LIN {X 0,Y 261.016,Z 653.466,A -85,B 0,C 180,E1 -18954.006,E2 -18954.006} C_VEL
LIN {X 0,Y 257.341,Z 662.24,A -85,B 0,C 180,E1 -18956.893,E2 -18956.893} C_VEL
LIN {X 0,Y 253.986,Z 670.002,A -85,B 0,C 180,E1 -18960.127,E2 -18960.127} C_VEL
LIN {X 0,Y 251.244,Z 676.279,A -85,B 0,C 180,E1 -18963.527,E2 -18963.527} C_VEL
LIN {X 0,Y 249.374,Z 680.762,A -85,B 0,C 180,E1 -18966.762,E2 -18966.762} C_VEL
LIN {X 0,Y 248.037,Z 684.043,A -85,B 0,C 180,E1 -18970.122,E2 -18970.122} C_VEL
LIN {X 0,Y 247.2,Z 686.071,A -85,B 0,C 180,E1 -18973.483,E2 -18973.483} C_VEL
LIN {X 0,Y 246.839,Z 686.909,A -85,B 0,C 180,E1 -18976.834,E2 -18976.834} C_VEL
LIN {X 0,Y 246.696,Z 686.594,A -85,B 0,C 180,E1 -18980.158,E2 -18980.158} C_VEL
LIN {X 0,Y 246.891,Z 685.135,A -85,B 0,C 180,E1 -18983.462,E2 -18983.462} C_VEL
LIN {X 0,Y 247.231,Z 682.514,A -85,B 0,C 180,E1 -18986.741,E2 -18986.741} C_VEL
LIN {X 0,Y 247.801,Z 678.647,A -85,B 0,C 180,E1 -18990,E2 -18990} C_VEL
LIN {X 0,Y 248.772,Z 673.495,A -85,B 0,C 180,E1 -18993.239,E2 -18993.239} C_VEL
LIN {X 0,Y 250.266,Z 666.931,A -85,B 0,C 180,E1 -18996.45,E2 -18996.45} C_VEL
LIN {X 0,Y 252.206,Z 659.844,A -85,B 0,C 180,E1 -18999.22,E2 -18999.22} C_VEL
LIN {X 0,Y 254.44,Z 651.357,A -85,B 0,C 180,E1 -19001.956,E2 -19001.956} C_VEL
LIN {X 0,Y 257.158,Z 641.157,A -85,B 0,C 180,E1 -19004.643,E2 -19004.643} C_VEL
LIN {X 0,Y 259.96,Z 630.71,A -85,B 0,C 180,E1 -19006.896,E2 -19006.896} C_VEL
LIN {X 0,Y 262.686,Z 619.377,A -85,B 0,C 180,E1 -19008.929,E2 -19008.929} C_VEL
LIN {X 0,Y 265.451,Z 607.068,A -85,B 0,C 180,E1 -19010.739,E2 -19010.739} C_VEL
LIN {X 0,Y 268.125,Z 593.612,A -85,B 0,C 180,E1 -19012.338,E2 -19012.338} C_VEL
LIN {X 0,Y 270.433,Z 579.688,A -85,B 0,C 180,E1 -19013.653,E2 -19013.653} C_VEL
LIN {X 0,Y 272.361,Z 565.38,A -85,B 0,C 180,E1 -19014.69,E2 -19014.69} C_VEL
LIN {X 0,Y 273.951,Z 549.877,A -85,B 0,C 180,E1 -19015.5,E2 -19015.5} C_VEL
LIN {X 0,Y 274.904,Z 534.682,A -85,B 0,C 180,E1 -19016.017,E2 -19016.017} C_VEL
LIN {X 0,Y 279.025,Z 439.219,A -85,B 0,C 180,E1 -19018.376,E2 -19018.376} C_VEL
LIN {X 0,Y 272.382,Z 423.601,A -85,B 0,C 180,E1 -19019.845,E2 -19019.845} C_VEL
LIN {X 0,Y 268.047,Z 414.836,A -85,B 0,C 180,E1 -19020.812,E2 -19020.812} C_VEL
LIN {X 0,Y 259.634,Z 400.449,A -85,B 0,C 180,E1 -19022.72,E2 -19022.72} C_VEL
LIN {X 0,Y 253.489,Z 390.868,A -85,B 0,C 180,E1 -19024.195,E2 -19024.195} C_VEL
LIN {X 0,Y 251.182,Z 387.293,A -85,B 0,C 180,E1 -19024.776,E2 -19024.776} C_VEL
LIN {X 0,Y 249.581,Z 385.053,A -85,B 0,C 180,E1 -19025.178,E2 -19025.178} C_VEL
LIN {X 0,Y 249.044,Z 383.079,A -85,B 0,C 180,E1 -19025.377,E2 -19025.377} C_VEL
LIN {X 0,Y 249.025,Z 383.091,A -85,B 0,C 180,E1 -19028.381,E2 -19028.381} C_VEL
LIN {X 0,Y 248.997,Z 383.093,A -85,B 0,C 180,E1 -19032.788,E2 -19032.788} C_VEL
LIN {X 0,Y 248.982,Z 383.08,A -85,B 0,C 180,E1 -19037.354,E2 -19037.354} C_VEL
LIN {X 0,Y 249.024,Z 383.085,A -85,B 0,C 180,E1 -19042.207,E2 -19042.207} C_VEL
LIN {X 0,Y 249.045,Z 383.078,A -85,B 0,C 180,E1 -19045.639,E2 -19045.639} C_VEL
LIN {X 0,Y 249.004,Z 383.09,A -85,B 0,C 180,E1 -19049.466,E2 -19049.466} C_VEL
LIN {X 0,Y 249.014,Z 383.029,A -85,B 0,C 180,E1 -19053.154,E2 -19053.154} C_VEL
LIN {X 0,Y 249.01,Z 383.065,A -85,B 0,C 180,E1 -19056.725,E2 -19056.725} C_VEL
LIN {X 0,Y 249.088,Z 383.08,A -85,B 0,C 180,E1 -19060.209,E2 -19060.209} C_VEL
LIN {X 0,Y 249.198,Z 383.054,A -85,B 0,C 180,E1 -19063.618,E2 -19063.618} C_VEL
LIN {X 0,Y 249.19,Z 383.049,A -85,B 0,C 180,E1 -19067.817,E2 -19067.817} C_VEL
LIN {X 0,Y 248.56,Z 383.129,A -85,B 0,C 180,E1 -19069.168,E2 -19069.168} C_VEL
LIN {X 0,Y 245.742,Z 383.496,A -85,B 0,C 180,E1 -19071.372,E2 -19071.372} C_VEL
LIN {X 0,Y 243.333,Z 383.789,A -85,B 0,C 180,E1 -19073.167,E2 -19073.167} C_VEL
LIN {X 0,Y 242.305,Z 383.906,A -85,B 0,C 180,E1 -19074.558,E2 -19074.558} C_VEL
LIN {X 0,Y 242.225,Z 383.914,A -85,B 0,C 180,E1 -19075.03,E2 -19075.03} C_VEL
LIN {X 0,Y 242.622,Z 383.886,A -85,B 0,C 180,E1 -19078.339,E2 -19078.339} C_VEL
LIN {X 0,Y 242.624,Z 383.866,A -85,B 0,C 180,E1 -19081.659,E2 -19081.659} C_VEL
LIN {X 0,Y 242.4,Z 383.906,A -85,B 0,C 180,E1 -19086.659,E2 -19086.659} C_VEL
LIN {X 0,Y 242.266,Z 383.931,A -85,B 0,C 180,E1 -19090.023,E2 -19090.023} C_VEL
LIN {X 0,Y 242.114,Z 383.946,A -85,B 0,C 180,E1 -19095.144,E2 -19095.144} C_VEL
LIN {X 0,Y 242.055,Z 383.945,A -85,B 0,C 180,E1 -19098.625,E2 -19098.625} C_VEL
LIN {X 0,Y 242.006,Z 383.951,A -85,B 0,C 180,E1 -19102.18,E2 -19102.18} C_VEL
LIN {X 0,Y 242.033,Z 383.952,A -85,B 0,C 180,E1 -19105.82,E2 -19105.82} C_VEL
LIN {X 0,Y 241.969,Z 383.963,A -85,B 0,C 180,E1 -19109.588,E2 -19109.588} C_VEL
LIN {X 0,Y 241.979,Z 383.964,A -85,B 0,C 180,E1 -19113.492,E2 -19113.492} C_VEL
LIN {X 0,Y 241.964,Z 383.967,A -85,B 0,C 180,E1 -19117.586,E2 -19117.586} C_VEL
LIN {X 0,Y 241.953,Z 384.049,A -85,B 0,C 180,E1 -19121.289,E2 -19121.289} C_VEL
LIN {X 0,Y 243.383,Z 388.779,A -85,B 0,C 180,E1 -19123.277,E2 -19123.277} C_VEL
LIN {X 0,Y 251.725,Z 403.288,A -85,B 0,C 180,E1 -19125.515,E2 -19125.515} C_VEL
LIN {X 0,Y 259.948,Z 419.151,A -85,B 0,C 180,E1 -19127.579,E2 -19127.579} C_VEL
LIN {X 0,Y 266.809,Z 434.583,A -85,B 0,C 180,E1 -19129.238,E2 -19129.238} C_VEL
LIN {X 0,Y 271.986,Z 447.57,A -85,B 0,C 180,E1 -19130.456,E2 -19130.456} C_VEL
LIN {X 0,Y 272.722,Z 452.165,A -85,B 0,C 180,E1 -19130.712,E2 -19130.712} C_VEL
LIN {X 0,Y 268.172,Z 555.027,A -85,B 0,C 180,E1 -19133.342,E2 -19133.342} C_VEL
LIN {X 0,Y 266.741,Z 570.811,A -85,B 0,C 180,E1 -19133.993,E2 -19133.993} C_VEL
LIN {X 0,Y 264.605,Z 586.544,A -85,B 0,C 180,E1 -19134.944,E2 -19134.944} C_VEL
LIN {X 0,Y 262.082,Z 601.542,A -85,B 0,C 180,E1 -19136.196,E2 -19136.196} C_VEL
LIN {X 0,Y 259.354,Z 615.018,A -85,B 0,C 180,E1 -19137.643,E2 -19137.643} C_VEL
LIN {X 0,Y 256.193,Z 628.75,A -85,B 0,C 180,E1 -19139.502,E2 -19139.502} C_VEL
LIN {X 0,Y 253.314,Z 640.146,A -85,B 0,C 180,E1 -19141.407,E2 -19141.407} C_VEL
LIN {X 0,Y 250.333,Z 651.665,A -85,B 0,C 180,E1 -19143.758,E2 -19143.758} C_VEL
LIN {X 0,Y 247.409,Z 662.845,A -85,B 0,C 180,E1 -19146.566,E2 -19146.566} C_VEL
LIN {X 0,Y 244.839,Z 672.073,A -85,B 0,C 180,E1 -19149.413,E2 -19149.413} C_VEL
LIN {X 0,Y 242.894,Z 679.934,A -85,B 0,C 180,E1 -19152.4,E2 -19152.4} C_VEL
LIN {X 0,Y 241.36,Z 686.864,A -85,B 0,C 180,E1 -19155.67,E2 -19155.67} C_VEL
LIN {X 0,Y 240.349,Z 692.458,A -85,B 0,C 180,E1 -19159.043,E2 -19159.043} C_VEL
LIN {X 0,Y 240.014,Z 695.768,A -85,B 0,C 180,E1 -19161.581,E2 -19161.581} C_VEL
LIN {X 0,Y 239.835,Z 699.127,A -85,B 0,C 180,E1 -19165.077,E2 -19165.077} C_VEL
LIN {X 0,Y 239.871,Z 701.027,A -85,B 0,C 180,E1 -19168.321,E2 -19168.321} C_VEL
LIN {X 0,Y 239.924,Z 701.581,A -85,B 0,C 180,E1 -19170,E2 -19170} C_VEL
LIN {X 0,Y 239.761,Z 701.819,A -85,B 0,C 180,E1 -19173.361,E2 -19173.361} C_VEL
LIN {X 0,Y 239.788,Z 700.928,A -85,B 0,C 180,E1 -19176.733,E2 -19176.733} C_VEL
LIN {X 0,Y 240.257,Z 698.904,A -85,B 0,C 180,E1 -19180.108,E2 -19180.108} C_VEL
LIN {X 0,Y 241.291,Z 695.662,A -85,B 0,C 180,E1 -19183.474,E2 -19183.474} C_VEL
LIN {X 0,Y 242.893,Z 691.191,A -85,B 0,C 180,E1 -19186.819,E2 -19186.819} C_VEL
LIN {X 0,Y 245.272,Z 685.389,A -85,B 0,C 180,E1 -19190.111,E2 -19190.111} C_VEL
LIN {X 0,Y 248.318,Z 678.108,A -85,B 0,C 180,E1 -19193.343,E2 -19193.343} C_VEL
LIN {X 0,Y 251.8,Z 670.353,A -85,B 0,C 180,E1 -19196.078,E2 -19196.078} C_VEL
LIN {X 0,Y 254.976,Z 662.549,A -85,B 0,C 180,E1 -19198.39,E2 -19198.39} C_VEL
LIN {X 0,Y 259.415,Z 651.682,A -85,B 0,C 180,E1 -19200.98,E2 -19200.98} C_VEL
LIN {X 0,Y 263.606,Z 640.549,A -85,B 0,C 180,E1 -19203.131,E2 -19203.131} C_VEL
LIN {X 0,Y 267.847,Z 628.357,A -85,B 0,C 180,E1 -19205.028,E2 -19205.028} C_VEL
LIN {X 0,Y 270.967,Z 618.154,A -85,B 0,C 180,E1 -19206.335,E2 -19206.335} C_VEL
LIN {X 0,Y 274.472,Z 605.361,A -85,B 0,C 180,E1 -19207.686,E2 -19207.686} C_VEL
LIN {X 0,Y 277.752,Z 590.92,A -85,B 0,C 180,E1 -19208.891,E2 -19208.891} C_VEL
LIN {X 0,Y 280.638,Z 575.825,A -85,B 0,C 180,E1 -19209.804,E2 -19209.804} C_VEL
LIN {X 0,Y 282.692,Z 560.992,A -85,B 0,C 180,E1 -19210.445,E2 -19210.445} C_VEL
LIN {X 0,Y 283.971,Z 544.545,A -85,B 0,C 180,E1 -19210.925,E2 -19210.925} C_VEL
LIN {X 0,Y 288.516,Z 461.824,A -85,B 0,C 180,E1 -19212.922,E2 -19212.922} C_VEL
LIN {X 0,Y 282.932,Z 449.608,A -85,B 0,C 180,E1 -19214.599,E2 -19214.599} C_VEL
LIN {X 0,Y 277.69,Z 439.213,A -85,B 0,C 180,E1 -19216.25,E2 -19216.25} C_VEL
LIN {X 0,Y 270.529,Z 426.425,A -85,B 0,C 180,E1 -19218.661,E2 -19218.661} C_VEL
LIN {X 0,Y 263.822,Z 415.704,A -85,B 0,C 180,E1 -19221.121,E2 -19221.121} C_VEL
LIN {X 0,Y 259.64,Z 409.46,A -85,B 0,C 180,E1 -19222.783,E2 -19222.783} C_VEL
LIN {X 0,Y 256.451,Z 404.711,A -85,B 0,C 180,E1 -19224.143,E2 -19224.143} C_VEL
LIN {X 0,Y 252.023,Z 398.57,A -85,B 0,C 180,E1 -19226.166,E2 -19226.166} C_VEL
LIN {X 0,Y 248.403,Z 393.715,A -85,B 0,C 180,E1 -19227.967,E2 -19227.967} C_VEL
LIN {X 0,Y 246.962,Z 391.993,A -85,B 0,C 180,E1 -19228.717,E2 -19228.717} C_VEL
LIN {X 0,Y 244,Z 388.202,A -85,B 0,C 180,E1 -19230.369,E2 -19230.369} C_VEL
LIN {X 0,Y 242.753,Z 386.342,A -85,B 0,C 180,E1 -19231.167,E2 -19231.167} C_VEL
LIN {X 0,Y 241.997,Z 383.957,A -85,B 0,C 180,E1 -19233.248,E2 -19233.248} C_VEL
LIN {X 0,Y 242.027,Z 383.957,A -85,B 0,C 180,E1 -19236.013,E2 -19236.013} C_VEL
LIN {X 0,Y 242.036,Z 383.955,A -85,B 0,C 180,E1 -19239.609,E2 -19239.609} C_VEL
LIN {X 0,Y 242.164,Z 383.937,A -85,B 0,C 180,E1 -19243.279,E2 -19243.279} C_VEL
LIN {X 0,Y 242.151,Z 383.942,A -85,B 0,C 180,E1 -19246.575,E2 -19246.575} C_VEL
LIN {X 0,Y 242.343,Z 383.918,A -85,B 0,C 180,E1 -19250.405,E2 -19250.405} C_VEL
LIN {X 0,Y 242.399,Z 383.915,A -85,B 0,C 180,E1 -19253.341,E2 -19253.341} C_VEL
LIN {X 0,Y 242.631,Z 383.882,A -85,B 0,C 180,E1 -19258.341,E2 -19258.341} C_VEL
LIN {X 0,Y 242.624,Z 383.889,A -85,B 0,C 180,E1 -19261.661,E2 -19261.661} C_VEL
LIN {X 0,Y 242.4,Z 383.906,A -85,B 0,C 180,E1 -19266.661,E2 -19266.661} C_VEL
LIN {X 0,Y 242.27,Z 383.926,A -85,B 0,C 180,E1 -19270.024,E2 -19270.024} C_VEL
LIN {X 0,Y 242.169,Z 383.935,A -85,B 0,C 180,E1 -19275.141,E2 -19275.141} C_VEL
LIN {X 0,Y 242.051,Z 383.922,A -85,B 0,C 180,E1 -19278.791,E2 -19278.791} C_VEL
LIN {X 0,Y 242.765,Z 386.257,A -85,B 0,C 180,E1 -19279.337,E2 -19279.337} C_VEL
LIN {X 0,Y 244.854,Z 388.758,A -85,B 0,C 180,E1 -19280.555,E2 -19280.555} C_VEL
LIN {X 0,Y 246.633,Z 389.798,A -85,B 0,C 180,E1 -19281.462,E2 -19281.462} C_VEL
LIN {X 0,Y 248.217,Z 392.799,A -85,B 0,C 180,E1 -19282.364,E2 -19282.364} C_VEL
LIN {X 0,Y 250.878,Z 395.128,A -85,B 0,C 180,E1 -19283.638,E2 -19283.638} C_VEL
LIN {X 0,Y 253.737,Z 399.159,A -85,B 0,C 180,E1 -19285.009,E2 -19285.009} C_VEL
LIN {X 0,Y 255.513,Z 400.971,A -85,B 0,C 180,E1 -19285.782,E2 -19285.782} C_VEL
LIN {X 0,Y 258.133,Z 404.484,A -85,B 0,C 180,E1 -19286.914,E2 -19286.914} C_VEL
LIN {X 0,Y 259.914,Z 406.69,A -85,B 0,C 180,E1 -19287.64,E2 -19287.64} C_VEL
LIN {X 0,Y 263.34,Z 411.23,A -85,B 0,C 180,E1 -19288.984,E2 -19288.984} C_VEL
LIN {X 0,Y 269.38,Z 419.469,A -85,B 0,C 180,E1 -19291.18,E2 -19291.18} C_VEL
LIN {X 0,Y 276.643,Z 430.325,A -85,B 0,C 180,E1 -19293.598,E2 -19293.598} C_VEL
LIN {X 0,Y 282.542,Z 440.74,A -85,B 0,C 180,E1 -19295.443,E2 -19295.443} C_VEL
LIN {X 0,Y 288.955,Z 453.487,A -85,B 0,C 180,E1 -19297.34,E2 -19297.34} C_VEL
LIN {X 0,Y 283.774,Z 541.587,A -85,B 0,C 180,E1 -19299.44,E2 -19299.44} C_VEL
LIN {X 0,Y 282.258,Z 556.763,A -85,B 0,C 180,E1 -19300.037,E2 -19300.037} C_VEL
LIN {X 0,Y 280.123,Z 570.776,A -85,B 0,C 180,E1 -19300.813,E2 -19300.813} C_VEL
LIN {X 0,Y 277.323,Z 585.198,A -85,B 0,C 180,E1 -19301.89,E2 -19301.89} C_VEL
LIN {X 0,Y 274.227,Z 597.838,A -85,B 0,C 180,E1 -19303.079,E2 -19303.079} C_VEL
LIN {X 0,Y 270.778,Z 610.647,A -85,B 0,C 180,E1 -19304.621,E2 -19304.621} C_VEL
LIN {X 0,Y 267.002,Z 622.242,A -85,B 0,C 180,E1 -19306.295,E2 -19306.295} C_VEL
LIN {X 0,Y 262.9,Z 633.747,A -85,B 0,C 180,E1 -19308.349,E2 -19308.349} C_VEL
LIN {X 0,Y 259.167,Z 643.251,A -85,B 0,C 180,E1 -19310.412,E2 -19310.412} C_VEL
LIN {X 0,Y 255.07,Z 653.132,A -85,B 0,C 180,E1 -19313.04,E2 -19313.04} C_VEL
LIN {X 0,Y 251.163,Z 661.982,A -85,B 0,C 180,E1 -19315.969,E2 -19315.969} C_VEL
LIN {X 0,Y 247.592,Z 669.859,A -85,B 0,C 180,E1 -19319.274,E2 -19319.274} C_VEL
LIN {X 0,Y 244.737,Z 676.055,A -85,B 0,C 180,E1 -19322.648,E2 -19322.648} C_VEL
LIN {X 0,Y 242.606,Z 680.758,A -85,B 0,C 180,E1 -19326.074,E2 -19326.074} C_VEL
LIN {X 0,Y 241.135,Z 684.108,A -85,B 0,C 180,E1 -19329.528,E2 -19329.528} C_VEL
LIN {X 0,Y 240.196,Z 686.207,A -85,B 0,C 180,E1 -19332.987,E2 -19332.987} C_VEL
LIN {X 0,Y 239.783,Z 687.114,A -85,B 0,C 180,E1 -19336.439,E2 -19336.439} C_VEL
LIN {X 0,Y 239.605,Z 686.867,A -85,B 0,C 180,E1 -19339.864,E2 -19339.864} C_VEL
LIN {X 0,Y 239.773,Z 685.477,A -85,B 0,C 180,E1 -19343.267,E2 -19343.267} C_VEL
LIN {X 0,Y 239.973,Z 684.337,A -85,B 0,C 180,E1 -19344.96,E2 -19344.96} C_VEL
LIN {X 0,Y 240.325,Z 681.149,A -85,B 0,C 180,E1 -19348.324,E2 -19348.324} C_VEL
LIN {X 0,Y 241.158,Z 676.72,A -85,B 0,C 180,E1 -19351.67,E2 -19351.67} C_VEL
LIN {X 0,Y 242.427,Z 670.96,A -85,B 0,C 180,E1 -19354.989,E2 -19354.989} C_VEL
LIN {X 0,Y 244.271,Z 663.702,A -85,B 0,C 180,E1 -19358.271,E2 -19358.271} C_VEL
LIN {X 0,Y 246.499,Z 655.924,A -85,B 0,C 180,E1 -19361.096,E2 -19361.096} C_VEL
LIN {X 0,Y 249.079,Z 646.608,A -85,B 0,C 180,E1 -19363.877,E2 -19363.877} C_VEL
LIN {X 0,Y 251.693,Z 637.137,A -85,B 0,C 180,E1 -19366.214,E2 -19366.214} C_VEL
LIN {X 0,Y 254.743,Z 625.879,A -85,B 0,C 180,E1 -19368.498,E2 -19368.498} C_VEL
LIN {X 0,Y 257.723,Z 613.535,A -85,B 0,C 180,E1 -19370.555,E2 -19370.555} C_VEL
LIN {X 0,Y 260.701,Z 599.893,A -85,B 0,C 180,E1 -19372.382,E2 -19372.382} C_VEL
LIN {X 0,Y 263.204,Z 586.496,A -85,B 0,C 180,E1 -19373.82,E2 -19373.82} C_VEL
LIN {X 0,Y 265.467,Z 571.622,A -85,B 0,C 180,E1 -19375.061,E2 -19375.061} C_VEL
LIN {X 0,Y 267.314,Z 556.746,A -85,B 0,C 180,E1 -19375.971,E2 -19375.971} C_VEL
LIN {X 0,Y 268.538,Z 541.777,A -85,B 0,C 180,E1 -19376.613,E2 -19376.613} C_VEL
LIN {X 0,Y 273.103,Z 442.016,A -85,B 0,C 180,E1 -19379.148,E2 -19379.148} C_VEL
LIN {X 0,Y 272.682,Z 440.051,A -85,B 0,C 180,E1 -19379.274,E2 -19379.274} C_VEL
LIN {X 0,Y 265.883,Z 424.291,A -85,B 0,C 180,E1 -19380.848,E2 -19380.848} C_VEL
LIN {X 0,Y 259.43,Z 412.346,A -85,B 0,C 180,E1 -19382.341,E2 -19382.341} C_VEL
LIN {X 0,Y 251.681,Z 399.57,A -85,B 0,C 180,E1 -19384.223,E2 -19384.223} C_VEL
LIN {X 0,Y 246.829,Z 392.184,A -85,B 0,C 180,E1 -19385.467,E2 -19385.467} C_VEL
LIN {X 0,Y 244.256,Z 388.333,A -85,B 0,C 180,E1 -19386.151,E2 -19386.151} C_VEL
LIN {X 0,Y 242.488,Z 385.859,A -85,B 0,C 180,E1 -19386.628,E2 -19386.628} C_VEL
LIN {X 0,Y 241.977,Z 383.956,A -85,B 0,C 180,E1 -19386.854,E2 -19386.854} C_VEL
LIN {X 0,Y 241.917,Z 383.957,A -85,B 0,C 180,E1 -19390.944,E2 -19390.944} C_VEL
LIN {X 0,Y 241.914,Z 383.967,A -85,B 0,C 180,E1 -19394.206,E2 -19394.206} C_VEL
LIN {X 0,Y 241.909,Z 383.97,A -85,B 0,C 180,E1 -19398.07,E2 -19398.07} C_VEL
LIN {X 0,Y 241.968,Z 383.965,A -85,B 0,C 180,E1 -19402.413,E2 -19402.413} C_VEL
LIN {X 0,Y 241.982,Z 383.959,A -85,B 0,C 180,E1 -19406.507,E2 -19406.507} C_VEL
LIN {X 0,Y 241.978,Z 383.947,A -85,B 0,C 180,E1 -19410.613,E2 -19410.613} C_VEL
LIN {X 0,Y 241.998,Z 383.901,A -85,B 0,C 180,E1 -19414.197,E2 -19414.197} C_VEL
LIN {X 0,Y 242.018,Z 383.96,A -85,B 0,C 180,E1 -19418.319,E2 -19418.319} C_VEL
LIN {X 0,Y 242.118,Z 383.933,A -85,B 0,C 180,E1 -19423.315,E2 -19423.315} C_VEL
LIN {X 0,Y 242.142,Z 383.927,A -85,B 0,C 180,E1 -19427.836,E2 -19427.836} C_VEL
LIN {X 0,Y 242.387,Z 383.916,A -85,B 0,C 180,E1 -19431.663,E2 -19431.663} C_VEL
LIN {X 0,Y 242.403,Z 383.903,A -85,B 0,C 180,E1 -19433.34,E2 -19433.34} C_VEL
LIN {X 0,Y 242.225,Z 383.914,A -85,B 0,C 180,E1 -19435.03,E2 -19435.03} C_VEL
LIN {X 0,Y 241.632,Z 383.999,A -85,B 0,C 180,E1 -19436.422,E2 -19436.422} C_VEL
LIN {X 0,Y 239.015,Z 384.335,A -85,B 0,C 180,E1 -19438.701,E2 -19438.701} C_VEL
LIN {X 0,Y 235.856,Z 384.71,A -85,B 0,C 180,E1 -19441.503,E2 -19441.503} C_VEL
LIN {X 0,Y 235.424,Z 384.765,A -85,B 0,C 180,E1 -19442.47,E2 -19442.47} C_VEL
LIN {X 0,Y 235.351,Z 384.782,A -85,B 0,C 180,E1 -19446.859,E2 -19446.859} C_VEL
LIN {X 0,Y 235.212,Z 384.809,A -85,B 0,C 180,E1 -19450.327,E2 -19450.327} C_VEL
LIN {X 0,Y 235.065,Z 384.827,A -85,B 0,C 180,E1 -19455.609,E2 -19455.609} C_VEL
LIN {X 0,Y 234.996,Z 384.828,A -85,B 0,C 180,E1 -19459.206,E2 -19459.206} C_VEL
LIN {X 0,Y 234.948,Z 384.831,A -85,B 0,C 180,E1 -19462.883,E2 -19462.883} C_VEL
LIN {X 0,Y 234.945,Z 384.835,A -85,B 0,C 180,E1 -19466.66,E2 -19466.66} C_VEL
LIN {X 0,Y 234.899,Z 384.846,A -85,B 0,C 180,E1 -19470.572,E2 -19470.572} C_VEL
LIN {X 0,Y 234.921,Z 384.848,A -85,B 0,C 180,E1 -19474.639,E2 -19474.639} C_VEL
LIN {X 0,Y 234.9,Z 384.831,A -85,B 0,C 180,E1 -19479.476,E2 -19479.476} C_VEL
LIN {X 0,Y 234.902,Z 384.921,A -85,B 0,C 180,E1 -19480.033,E2 -19480.033} C_VEL
LIN {X 0,Y 236.055,Z 388.638,A -85,B 0,C 180,E1 -19481.632,E2 -19481.632} C_VEL
LIN {X 0,Y 242.869,Z 400.164,A -85,B 0,C 180,E1 -19483.614,E2 -19483.614} C_VEL
LIN {X 0,Y 248.037,Z 409.511,A -85,B 0,C 180,E1 -19485.029,E2 -19485.029} C_VEL
LIN {X 0,Y 255.154,Z 423.383,A -85,B 0,C 180,E1 -19486.88,E2 -19486.88} C_VEL
LIN {X 0,Y 261.861,Z 438.74,A -85,B 0,C 180,E1 -19488.573,E2 -19488.573} C_VEL
LIN {X 0,Y 266.476,Z 450.566,A -85,B 0,C 180,E1 -19489.711,E2 -19489.711} C_VEL
LIN {X 0,Y 266.886,Z 454.888,A -85,B 0,C 180,E1 -19489.916,E2 -19489.916} C_VEL
LIN {X 0,Y 262.175,Z 555.901,A -85,B 0,C 180,E1 -19492.542,E2 -19492.542} C_VEL
LIN {X 0,Y 260.688,Z 571.263,A -85,B 0,C 180,E1 -19493.201,E2 -19493.201} C_VEL
LIN {X 0,Y 258.577,Z 586.173,A -85,B 0,C 180,E1 -19494.122,E2 -19494.122} C_VEL
LIN {X 0,Y 256.163,Z 600.234,A -85,B 0,C 180,E1 -19495.304,E2 -19495.304} C_VEL
LIN {X 0,Y 253.337,Z 613.909,A -85,B 0,C 180,E1 -19496.777,E2 -19496.777} C_VEL
LIN {X 0,Y 250.012,Z 627.824,A -85,B 0,C 180,E1 -19498.664,E2 -19498.664} C_VEL
LIN {X 0,Y 247.101,Z 639.327,A -85,B 0,C 180,E1 -19500.618,E2 -19500.618} C_VEL
LIN {X 0,Y 243.909,Z 650.749,A -85,B 0,C 180,E1 -19502.964,E2 -19502.964} C_VEL
LIN {X 0,Y 241.231,Z 660.698,A -85,B 0,C 180,E1 -19505.471,E2 -19505.471} C_VEL
LIN {X 0,Y 238.461,Z 670.255,A -85,B 0,C 180,E1 -19508.383,E2 -19508.383} C_VEL
LIN {X 0,Y 236.36,Z 678.203,A -85,B 0,C 180,E1 -19511.358,E2 -19511.358} C_VEL
LIN {X 0,Y 234.752,Z 684.78,A -85,B 0,C 180,E1 -19514.369,E2 -19514.369} C_VEL
LIN {X 0,Y 233.503,Z 690.802,A -85,B 0,C 180,E1 -19517.837,E2 -19517.837} C_VEL
LIN {X 0,Y 232.941,Z 695.426,A -85,B 0,C 180,E1 -19521.323,E2 -19521.323} C_VEL
LIN {X 0,Y 232.74,Z 698.718,A -85,B 0,C 180,E1 -19524.802,E2 -19524.802} C_VEL
LIN {X 0,Y 232.78,Z 700.754,A -85,B 0,C 180,E1 -19528.27,E2 -19528.27} C_VEL
LIN {X 0,Y 232.855,Z 701.33,A -85,B 0,C 180,E1 -19530,E2 -19530} C_VEL
LIN {X 0,Y 232.667,Z 701.61,A -85,B 0,C 180,E1 -19533.463,E2 -19533.463} C_VEL
LIN {X 0,Y 232.728,Z 700.763,A -85,B 0,C 180,E1 -19536.938,E2 -19536.938} C_VEL
LIN {X 0,Y 233.207,Z 698.766,A -85,B 0,C 180,E1 -19540.417,E2 -19540.417} C_VEL
LIN {X 0,Y 234.322,Z 695.565,A -85,B 0,C 180,E1 -19543.883,E2 -19543.883} C_VEL
LIN {X 0,Y 236.037,Z 691.144,A -85,B 0,C 180,E1 -19547.322,E2 -19547.322} C_VEL
LIN {X 0,Y 238.553,Z 685.395,A -85,B 0,C 180,E1 -19550.703,E2 -19550.703} C_VEL
LIN {X 0,Y 241.776,Z 678.17,A -85,B 0,C 180,E1 -19554.014,E2 -19554.014} C_VEL
LIN {X 0,Y 245.407,Z 670.478,A -85,B 0,C 180,E1 -19556.811,E2 -19556.811} C_VEL
LIN {X 0,Y 248.735,Z 662.714,A -85,B 0,C 180,E1 -19559.17,E2 -19559.17} C_VEL
LIN {X 0,Y 253.353,Z 651.94,A -85,B 0,C 180,E1 -19561.807,E2 -19561.807} C_VEL
LIN {X 0,Y 258.082,Z 639.885,A -85,B 0,C 180,E1 -19564.17,E2 -19564.17} C_VEL
LIN {X 0,Y 262.542,Z 627.618,A -85,B 0,C 180,E1 -19566.08,E2 -19566.08} C_VEL
LIN {X 0,Y 266.617,Z 614.433,A -85,B 0,C 180,E1 -19567.749,E2 -19567.749} C_VEL
LIN {X 0,Y 270.291,Z 600.901,A -85,B 0,C 180,E1 -19569.09,E2 -19569.09} C_VEL
LIN {X 0,Y 273.31,Z 587.513,A -85,B 0,C 180,E1 -19570.126,E2 -19570.126} C_VEL
LIN {X 0,Y 276.02,Z 572.821,A -85,B 0,C 180,E1 -19570.969,E2 -19570.969} C_VEL
LIN {X 0,Y 277.999,Z 557.747,A -85,B 0,C 180,E1 -19571.576,E2 -19571.576} C_VEL
LIN {X 0,Y 279.367,Z 537.905,A -85,B 0,C 180,E1 -19572.113,E2 -19572.113} C_VEL
LIN {X 0,Y 283.529,Z 464.298,A -85,B 0,C 180,E1 -19573.914,E2 -19573.914} C_VEL
LIN {X 0,Y 277.3,Z 450.617,A -85,B 0,C 180,E1 -19575.894,E2 -19575.894} C_VEL
LIN {X 0,Y 270.168,Z 437.023,A -85,B 0,C 180,E1 -19578.304,E2 -19578.304} C_VEL
LIN {X 0,Y 264.136,Z 426.624,A -85,B 0,C 180,E1 -19580.515,E2 -19580.515} C_VEL
LIN {X 0,Y 259.555,Z 419.395,A -85,B 0,C 180,E1 -19582.319,E2 -19582.319} C_VEL
LIN {X 0,Y 254.001,Z 410.857,A -85,B 0,C 180,E1 -19584.719,E2 -19584.719} C_VEL
LIN {X 0,Y 249.5,Z 404.514,A -85,B 0,C 180,E1 -19586.852,E2 -19586.852} C_VEL
LIN {X 0,Y 245.915,Z 399.512,A -85,B 0,C 180,E1 -19588.718,E2 -19588.718} C_VEL
LIN {X 0,Y 241.967,Z 394.584,A -85,B 0,C 180,E1 -19590.958,E2 -19590.958} C_VEL
LIN {X 0,Y 240.299,Z 392.365,A -85,B 0,C 180,E1 -19592.003,E2 -19592.003} C_VEL
LIN {X 0,Y 237.735,Z 389.626,A -85,B 0,C 180,E1 -19593.677,E2 -19593.677} C_VEL
LIN {X 0,Y 235.764,Z 387.295,A -85,B 0,C 180,E1 -19595.099,E2 -19595.099} C_VEL
LIN {X 0,Y 235.14,Z 385.645,A -85,B 0,C 180,E1 -19595.735,E2 -19595.735} C_VEL
LIN {X 0,Y 234.95,Z 384.834,A -85,B 0,C 180,E1 -19596.651,E2 -19596.651} C_VEL
LIN {X 0,Y 235.008,Z 384.826,A -85,B 0,C 180,E1 -19600.795,E2 -19600.795} C_VEL
LIN {X 0,Y 235.115,Z 384.812,A -85,B 0,C 180,E1 -19604.394,E2 -19604.394} C_VEL
LIN {X 0,Y 235.29,Z 384.798,A -85,B 0,C 180,E1 -19610.298,E2 -19610.298} C_VEL
LIN {X 0,Y 235.35,Z 384.79,A -85,B 0,C 180,E1 -19613.141,E2 -19613.141} C_VEL
LIN {X 0,Y 235.59,Z 384.759,A -85,B 0,C 180,E1 -19618.291,E2 -19618.291} C_VEL
LIN {X 0,Y 235.582,Z 384.766,A -85,B 0,C 180,E1 -19621.71,E2 -19621.71} C_VEL
LIN {X 0,Y 235.351,Z 384.783,A -85,B 0,C 180,E1 -19626.861,E2 -19626.861} C_VEL
LIN {X 0,Y 235.216,Z 384.802,A -85,B 0,C 180,E1 -19630.328,E2 -19630.328} C_VEL
LIN {X 0,Y 235.107,Z 384.839,A -85,B 0,C 180,E1 -19634.72,E2 -19634.72} C_VEL
LIN {X 0,Y 235.883,Z 387.265,A -85,B 0,C 180,E1 -19635.444,E2 -19635.444} C_VEL
LIN {X 0,Y 237.841,Z 389.581,A -85,B 0,C 180,E1 -19636.851,E2 -19636.851} C_VEL
LIN {X 0,Y 239.988,Z 390.881,A -85,B 0,C 180,E1 -19638.185,E2 -19638.185} C_VEL
LIN {X 0,Y 241.524,Z 393.744,A -85,B 0,C 180,E1 -19639.22,E2 -19639.22} C_VEL
LIN {X 0,Y 243.788,Z 395.899,A -85,B 0,C 180,E1 -19640.513,E2 -19640.513} C_VEL
LIN {X 0,Y 244.648,Z 396.748,A -85,B 0,C 180,E1 -19640.983,E2 -19640.983} C_VEL
LIN {X 0,Y 246.783,Z 399.953,A -85,B 0,C 180,E1 -19642.17,E2 -19642.17} C_VEL
LIN {X 0,Y 249.027,Z 402.068,A -85,B 0,C 180,E1 -19643.273,E2 -19643.273} C_VEL
LIN {X 0,Y 251.734,Z 405.737,A -85,B 0,C 180,E1 -19644.593,E2 -19644.593} C_VEL
LIN {X 0,Y 253.077,Z 407.19,A -85,B 0,C 180,E1 -19645.198,E2 -19645.198} C_VEL
LIN {X 0,Y 256.165,Z 411.153,A -85,B 0,C 180,E1 -19646.559,E2 -19646.559} C_VEL
LIN {X 0,Y 260.587,Z 417.195,A -85,B 0,C 180,E1 -19648.383,E2 -19648.383} C_VEL
LIN {X 0,Y 266.466,Z 425.351,A -85,B 0,C 180,E1 -19650.595,E2 -19650.595} C_VEL
LIN {X 0,Y 273.428,Z 435.98,A -85,B 0,C 180,E1 -19652.998,E2 -19652.998} C_VEL
LIN {X 0,Y 279.462,Z 446.954,A -85,B 0,C 180,E1 -19654.954,E2 -19654.954} C_VEL
LIN {X 0,Y 283.996,Z 456.118,A -85,B 0,C 180,E1 -19656.354,E2 -19656.354} C_VEL
LIN {X 0,Y 279.169,Z 535.328,A -85,B 0,C 180,E1 -19658.219,E2 -19658.219} C_VEL
LIN {X 0,Y 277.915,Z 551.497,A -85,B 0,C 180,E1 -19658.777,E2 -19658.777} C_VEL
LIN {X 0,Y 275.861,Z 566.051,A -85,B 0,C 180,E1 -19659.486,E2 -19659.486} C_VEL
LIN {X 0,Y 273.179,Z 580.638,A -85,B 0,C 180,E1 -19660.488,E2 -19660.488} C_VEL
LIN {X 0,Y 269.715,Z 595.073,A -85,B 0,C 180,E1 -19661.765,E2 -19661.765} C_VEL
LIN {X 0,Y 265.811,Z 609.298,A -85,B 0,C 180,E1 -19663.429,E2 -19663.429} C_VEL
LIN {X 0,Y 261.751,Z 621.543,A -85,B 0,C 180,E1 -19665.186,E2 -19665.186} C_VEL
LIN {X 0,Y 257.441,Z 633.224,A -85,B 0,C 180,E1 -19667.27,E2 -19667.27} C_VEL
LIN {X 0,Y 253.52,Z 642.766,A -85,B 0,C 180,E1 -19669.348,E2 -19669.348} C_VEL
LIN {X 0,Y 249.618,Z 651.776,A -85,B 0,C 180,E1 -19671.727,E2 -19671.727} C_VEL
LIN {X 0,Y 245.595,Z 660.581,A -85,B 0,C 180,E1 -19674.586,E2 -19674.586} C_VEL
LIN {X 0,Y 241.851,Z 668.409,A -85,B 0,C 180,E1 -19677.78,E2 -19677.78} C_VEL
LIN {X 0,Y 238.877,Z 674.526,A -85,B 0,C 180,E1 -19680.958,E2 -19680.958} C_VEL
LIN {X 0,Y 236.37,Z 679.677,A -85,B 0,C 180,E1 -19684.461,E2 -19684.461} C_VEL
LIN {X 0,Y 234.494,Z 683.683,A -85,B 0,C 180,E1 -19688.297,E2 -19688.297} C_VEL
LIN {X 0,Y 233.649,Z 685.412,A -85,B 0,C 180,E1 -19690.678,E2 -19690.678} C_VEL
LIN {X 0,Y 232.923,Z 686.978,A -85,B 0,C 180,E1 -19694.243,E2 -19694.243} C_VEL
LIN {X 0,Y 232.577,Z 687.373,A -85,B 0,C 180,E1 -19697.788,E2 -19697.788} C_VEL
LIN {X 0,Y 232.548,Z 686.622,A -85,B 0,C 180,E1 -19701.309,E2 -19701.309} C_VEL
LIN {X 0,Y 232.904,Z 684.678,A -85,B 0,C 180,E1 -19704.806,E2 -19704.806} C_VEL
LIN {X 0,Y 233.231,Z 681.558,A -85,B 0,C 180,E1 -19708.273,E2 -19708.273} C_VEL
LIN {X 0,Y 234.09,Z 677.201,A -85,B 0,C 180,E1 -19711.721,E2 -19711.721} C_VEL
LIN {X 0,Y 235.395,Z 671.517,A -85,B 0,C 180,E1 -19715.139,E2 -19715.139} C_VEL
LIN {X 0,Y 237.276,Z 664.345,A -85,B 0,C 180,E1 -19718.517,E2 -19718.517} C_VEL
LIN {X 0,Y 239.578,Z 656.658,A -85,B 0,C 180,E1 -19721.421,E2 -19721.421} C_VEL
LIN {X 0,Y 242.244,Z 647.445,A -85,B 0,C 180,E1 -19724.277,E2 -19724.277} C_VEL
LIN {X 0,Y 244.93,Z 638.097,A -85,B 0,C 180,E1 -19726.675,E2 -19726.675} C_VEL
LIN {X 0,Y 248.082,Z 626.975,A -85,B 0,C 180,E1 -19729.013,E2 -19729.013} C_VEL
LIN {X 0,Y 251.154,Z 614.801,A -85,B 0,C 180,E1 -19731.117,E2 -19731.117} C_VEL
LIN {X 0,Y 254.21,Z 601.412,A -85,B 0,C 180,E1 -19732.986,E2 -19732.986} C_VEL
LIN {X 0,Y 256.793,Z 588.264,A -85,B 0,C 180,E1 -19734.453,E2 -19734.453} C_VEL
LIN {X 0,Y 259.143,Z 573.85,A -85,B 0,C 180,E1 -19735.717,E2 -19735.717} C_VEL
LIN {X 0,Y 261.212,Z 558.129,A -85,B 0,C 180,E1 -19736.733,E2 -19736.733} C_VEL
LIN {X 0,Y 262.59,Z 542.125,A -85,B 0,C 180,E1 -19737.442,E2 -19737.442} C_VEL
LIN {X 0,Y 267.264,Z 444.023,A -85,B 0,C 180,E1 -19739.975,E2 -19739.975} C_VEL
LIN {X 0,Y 266.953,Z 442.33,A -85,B 0,C 180,E1 -19740.08,E2 -19740.08} C_VEL
LIN {X 0,Y 259.971,Z 426.154,A -85,B 0,C 180,E1 -19741.769,E2 -19741.769} C_VEL
LIN {X 0,Y 250.87,Z 410.085,A -85,B 0,C 180,E1 -19743.992,E2 -19743.992} C_VEL
LIN {X 0,Y 243.022,Z 397.668,A -85,B 0,C 180,E1 -19746.048,E2 -19746.048} C_VEL
LIN {X 0,Y 239.687,Z 392.871,A -85,B 0,C 180,E1 -19746.963,E2 -19746.963} C_VEL
LIN {X 0,Y 237.466,Z 389.416,A -85,B 0,C 180,E1 -19747.604,E2 -19747.604} C_VEL
LIN {X 0,Y 235.634,Z 387.109,A -85,B 0,C 180,E1 -19748.126,E2 -19748.126} C_VEL
LIN {X 0,Y 234.954,Z 384.844,A -85,B 0,C 180,E1 -19748.388,E2 -19748.388} C_VEL
LIN {X 0,Y 234.875,Z 384.853,A -85,B 0,C 180,E1 -19753.489,E2 -19753.489} C_VEL
LIN {X 0,Y 234.859,Z 384.831,A -85,B 0,C 180,E1 -19756.506,E2 -19756.506} C_VEL
LIN {X 0,Y 234.921,Z 384.836,A -85,B 0,C 180,E1 -19761.078,E2 -19761.078} C_VEL
LIN {X 0,Y 234.925,Z 384.837,A -85,B 0,C 180,E1 -19765.36,E2 -19765.36} C_VEL
LIN {X 0,Y 234.901,Z 384.847,A -85,B 0,C 180,E1 -19769.427,E2 -19769.427} C_VEL
LIN {X 0,Y 234.942,Z 384.778,A -85,B 0,C 180,E1 -19773.821,E2 -19773.821} C_VEL
LIN {X 0,Y 234.988,Z 384.838,A -85,B 0,C 180,E1 -19778.967,E2 -19778.967} C_VEL
LIN {X 0,Y 235.059,Z 384.811,A -85,B 0,C 180,E1 -19783.091,E2 -19783.091} C_VEL
LIN {X 0,Y 235.103,Z 384.803,A -85,B 0,C 180,E1 -19787.921,E2 -19787.921} C_VEL
LIN {X 0,Y 235.321,Z 384.794,A -85,B 0,C 180,E1 -19791.411,E2 -19791.411} C_VEL
LIN {X 0,Y 235.355,Z 384.783,A -85,B 0,C 180,E1 -19793.139,E2 -19793.139} C_VEL
LIN {X 0,Y 235.581,Z 384.764,A -85,B 0,C 180,E1 -19798.29,E2 -19798.29} C_VEL
LIN {X 0,Y 235.583,Z 384.743,A -85,B 0,C 180,E1 -19801.709,E2 -19801.709} C_VEL
LIN {X 0,Y 235.424,Z 384.765,A -85,B 0,C 180,E1 -19802.47,E2 -19802.47} C_VEL
LIN {X 0,Y 234.602,Z 384.883,A -85,B 0,C 180,E1 -19803.896,E2 -19803.896} C_VEL
LIN {X 0,Y 231.759,Z 385.237,A -85,B 0,C 180,E1 -19806.227,E2 -19806.227} C_VEL
LIN {X 0,Y 228.577,Z 385.634,A -85,B 0,C 180,E1 -19809.101,E2 -19809.101} C_VEL
LIN {X 0,Y 228.194,Z 385.681,A -85,B 0,C 180,E1 -19810.095,E2 -19810.095} C_VEL
LIN {X 0,Y 227.999,Z 385.698,A -85,B 0,C 180,E1 -19814.276,E2 -19814.276} C_VEL
LIN {X 0,Y 227.957,Z 385.698,A -85,B 0,C 180,E1 -19817.956,E2 -19817.956} C_VEL
LIN {X 0,Y 227.923,Z 385.705,A -85,B 0,C 180,E1 -19822.323,E2 -19822.323} C_VEL
LIN {X 0,Y 227.923,Z 385.709,A -85,B 0,C 180,E1 -19826.591,E2 -19826.591} C_VEL
LIN {X 0,Y 227.874,Z 385.719,A -85,B 0,C 180,E1 -19830.28,E2 -19830.28} C_VEL
LIN {X 0,Y 227.875,Z 385.721,A -85,B 0,C 180,E1 -19833.72,E2 -19833.72} C_VEL
LIN {X 0,Y 227.867,Z 385.71,A -85,B 0,C 180,E1 -19838.576,E2 -19838.576} C_VEL
LIN {X 0,Y 228.743,Z 388.344,A -85,B 0,C 180,E1 -19839.828,E2 -19839.828} C_VEL
LIN {X 0,Y 230.719,Z 391.843,A -85,B 0,C 180,E1 -19840.481,E2 -19840.481} C_VEL
LIN {X 0,Y 235.516,Z 399.555,A -85,B 0,C 180,E1 -19841.96,E2 -19841.96} C_VEL
LIN {X 0,Y 242.651,Z 412.162,A -85,B 0,C 180,E1 -19844.036,E2 -19844.036} C_VEL
LIN {X 0,Y 250.36,Z 427.498,A -85,B 0,C 180,E1 -19846.144,E2 -19846.144} C_VEL
LIN {X 0,Y 256.832,Z 442.496,A -85,B 0,C 180,E1 -19847.85,E2 -19847.85} C_VEL
LIN {X 0,Y 261.01,Z 453.476,A -85,B 0,C 180,E1 -19848.931,E2 -19848.931} C_VEL
LIN {X 0,Y 261.057,Z 457.73,A -85,B 0,C 180,E1 -19849.083,E2 -19849.083} C_VEL
LIN {X 0,Y 256.304,Z 555.345,A -85,B 0,C 180,E1 -19851.655,E2 -19851.655} C_VEL
LIN {X 0,Y 254.787,Z 570.836,A -85,B 0,C 180,E1 -19852.327,E2 -19852.327} C_VEL
LIN {X 0,Y 252.577,Z 585.791,A -85,B 0,C 180,E1 -19853.256,E2 -19853.256} C_VEL
LIN {X 0,Y 250.142,Z 599.644,A -85,B 0,C 180,E1 -19854.437,E2 -19854.437} C_VEL
LIN {X 0,Y 247.375,Z 612.792,A -85,B 0,C 180,E1 -19855.868,E2 -19855.868} C_VEL
LIN {X 0,Y 244.3,Z 625.57,A -85,B 0,C 180,E1 -19857.601,E2 -19857.601} C_VEL
LIN {X 0,Y 241.186,Z 637.415,A -85,B 0,C 180,E1 -19859.582,E2 -19859.582} C_VEL
LIN {X 0,Y 237.966,Z 648.387,A -85,B 0,C 180,E1 -19861.801,E2 -19861.801} C_VEL
LIN {X 0,Y 235.119,Z 658.54,A -85,B 0,C 180,E1 -19864.315,E2 -19864.315} C_VEL
LIN {X 0,Y 232.558,Z 667.157,A -85,B 0,C 180,E1 -19866.867,E2 -19866.867} C_VEL
LIN {X 0,Y 230.116,Z 675.58,A -85,B 0,C 180,E1 -19869.904,E2 -19869.904} C_VEL
LIN {X 0,Y 228.148,Z 682.919,A -85,B 0,C 180,E1 -19873.168,E2 -19873.168} C_VEL
LIN {X 0,Y 226.813,Z 689.005,A -85,B 0,C 180,E1 -19876.562,E2 -19876.562} C_VEL
LIN {X 0,Y 225.979,Z 693.998,A -85,B 0,C 180,E1 -19880.151,E2 -19880.151} C_VEL
LIN {X 0,Y 225.7,Z 696.898,A -85,B 0,C 180,E1 -19882.845,E2 -19882.845} C_VEL
LIN {X 0,Y 225.617,Z 699.587,A -85,B 0,C 180,E1 -19886.428,E2 -19886.428} C_VEL
LIN {X 0,Y 225.765,Z 701.078,A -85,B 0,C 180,E1 -19890,E2 -19890} C_VEL
LIN {X 0,Y 225.575,Z 701.401,A -85,B 0,C 180,E1 -19893.572,E2 -19893.572} C_VEL
LIN {X 0,Y 225.64,Z 700.598,A -85,B 0,C 180,E1 -19897.157,E2 -19897.157} C_VEL
LIN {X 0,Y 226.174,Z 698.624,A -85,B 0,C 180,E1 -19900.745,E2 -19900.745} C_VEL
LIN {X 0,Y 227.375,Z 695.469,A -85,B 0,C 180,E1 -19904.316,E2 -19904.316} C_VEL
LIN {X 0,Y 229.183,Z 691.097,A -85,B 0,C 180,E1 -19907.858,E2 -19907.858} C_VEL
LIN {X 0,Y 231.88,Z 685.4,A -85,B 0,C 180,E1 -19911.328,E2 -19911.328} C_VEL
LIN {X 0,Y 235.272,Z 678.231,A -85,B 0,C 180,E1 -19914.721,E2 -19914.721} C_VEL
LIN {X 0,Y 239.042,Z 670.605,A -85,B 0,C 180,E1 -19917.585,E2 -19917.585} C_VEL
LIN {X 0,Y 242.532,Z 662.879,A -85,B 0,C 180,E1 -19919.991,E2 -19919.991} C_VEL
LIN {X 0,Y 246.618,Z 653.811,A -85,B 0,C 180,E1 -19922.298,E2 -19922.298} C_VEL
LIN {X 0,Y 251.073,Z 643.162,A -85,B 0,C 180,E1 -19924.53,E2 -19924.53} C_VEL
LIN {X 0,Y 255.958,Z 630.422,A -85,B 0,C 180,E1 -19926.67,E2 -19926.67} C_VEL
LIN {X 0,Y 259.872,Z 618.835,A -85,B 0,C 180,E1 -19928.246,E2 -19928.246} C_VEL
LIN {X 0,Y 263.922,Z 605.192,A -85,B 0,C 180,E1 -19929.725,E2 -19929.725} C_VEL
LIN {X 0,Y 267.451,Z 590.824,A -85,B 0,C 180,E1 -19930.942,E2 -19930.942} C_VEL
LIN {X 0,Y 270.487,Z 575.854,A -85,B 0,C 180,E1 -19931.869,E2 -19931.869} C_VEL
LIN {X 0,Y 272.682,Z 561.245,A -85,B 0,C 180,E1 -19932.513,E2 -19932.513} C_VEL
LIN {X 0,Y 274.03,Z 545.206,A -85,B 0,C 180,E1 -19933.004,E2 -19933.004} C_VEL
LIN {X 0,Y 278.717,Z 467.006,A -85,B 0,C 180,E1 -19934.913,E2 -19934.913} C_VEL
LIN {X 0,Y 272.527,Z 453.399,A -85,B 0,C 180,E1 -19936.985,E2 -19936.985} C_VEL
LIN {X 0,Y 265.828,Z 440.511,A -85,B 0,C 180,E1 -19939.379,E2 -19939.379} C_VEL
LIN {X 0,Y 260.046,Z 430.56,A -85,B 0,C 180,E1 -19941.613,E2 -19941.613} C_VEL
LIN {X 0,Y 254.724,Z 421.952,A -85,B 0,C 180,E1 -19943.861,E2 -19943.861} C_VEL
LIN {X 0,Y 250.697,Z 415.829,A -85,B 0,C 180,E1 -19945.716,E2 -19945.716} C_VEL
LIN {X 0,Y 246.692,Z 410.025,A -85,B 0,C 180,E1 -19947.718,E2 -19947.718} C_VEL
LIN {X 0,Y 242.891,Z 404.752,A -85,B 0,C 180,E1 -19949.801,E2 -19949.801} C_VEL
LIN {X 0,Y 239.785,Z 400.627,A -85,B 0,C 180,E1 -19951.676,E2 -19951.676} C_VEL
LIN {X 0,Y 238.096,Z 398.486,A -85,B 0,C 180,E1 -19952.773,E2 -19952.773} C_VEL
LIN {X 0,Y 236.025,Z 396.228,A -85,B 0,C 180,E1 -19954.184,E2 -19954.184} C_VEL
LIN {X 0,Y 233.918,Z 393.568,A -85,B 0,C 180,E1 -19955.777,E2 -19955.777} C_VEL
LIN {X 0,Y 232.897,Z 391.613,A -85,B 0,C 180,E1 -19956.668,E2 -19956.668} C_VEL
LIN {X 0,Y 230.02,Z 389.905,A -85,B 0,C 180,E1 -19959.079,E2 -19959.079} C_VEL
LIN {X 0,Y 228.468,Z 387.598,A -85,B 0,C 180,E1 -19960.749,E2 -19960.749} C_VEL
LIN {X 0,Y 227.976,Z 385.706,A -85,B 0,C 180,E1 -19961.58,E2 -19961.58} C_VEL
LIN {X 0,Y 228.058,Z 385.702,A -85,B 0,C 180,E1 -19965.728,E2 -19965.728} C_VEL
LIN {X 0,Y 228.253,Z 385.666,A -85,B 0,C 180,E1 -19971.145,E2 -19971.145} C_VEL
LIN {X 0,Y 228.303,Z 385.665,A -85,B 0,C 180,E1 -19972.928,E2 -19972.928} C_VEL
LIN {X 0,Y 228.549,Z 385.636,A -85,B 0,C 180,E1 -19978.239,E2 -19978.239} C_VEL
LIN {X 0,Y 228.54,Z 385.643,A -85,B 0,C 180,E1 -19981.763,E2 -19981.763} C_VEL
LIN {X 0,Y 228.303,Z 385.66,A -85,B 0,C 180,E1 -19987.074,E2 -19987.074} C_VEL
LIN {X 0,Y 228.29,Z 385.848,A -85,B 0,C 180,E1 -19989.327,E2 -19989.327} C_VEL
LIN {X 0,Y 228.998,Z 388.224,A -85,B 0,C 180,E1 -19990.292,E2 -19990.292} C_VEL
LIN {X 0,Y 230.79,Z 390.441,A -85,B 0,C 180,E1 -19992.085,E2 -19992.085} C_VEL
LIN {X 0,Y 233.376,Z 391.871,A -85,B 0,C 180,E1 -19994.164,E2 -19994.164} C_VEL
LIN {X 0,Y 234.694,Z 394.627,A -85,B 0,C 180,E1 -19995.302,E2 -19995.302} C_VEL
LIN {X 0,Y 237.218,Z 396.964,A -85,B 0,C 180,E1 -19997.065,E2 -19997.065} C_VEL
LIN {X 0,Y 238.182,Z 397.77,A -85,B 0,C 180,E1 -19997.689,E2 -19997.689} C_VEL
LIN {X 0,Y 240.304,Z 401.058,A -85,B 0,C 180,E1 -19999.099,E2 -19999.099} C_VEL
LIN {X 0,Y 242.558,Z 403.179,A -85,B 0,C 180,E1 -20000.399,E2 -20000.399} C_VEL
LIN {X 0,Y 245.003,Z 406.646,A -85,B 0,C 180,E1 -20001.785,E2 -20001.785} C_VEL
LIN {X 0,Y 246.939,Z 408.673,A -85,B 0,C 180,E1 -20002.775,E2 -20002.775} C_VEL
LIN {X 0,Y 249.836,Z 412.382,A -85,B 0,C 180,E1 -20004.211,E2 -20004.211} C_VEL
LIN {X 0,Y 254.682,Z 418.749,A -85,B 0,C 180,E1 -20006.422,E2 -20006.422} C_VEL
LIN {X 0,Y 258.287,Z 423.722,A -85,B 0,C 180,E1 -20007.939,E2 -20007.939} C_VEL
LIN {X 0,Y 265.365,Z 433.841,A -85,B 0,C 180,E1 -20010.653,E2 -20010.653} C_VEL
LIN {X 0,Y 271.504,Z 443.913,A -85,B 0,C 180,E1 -20012.819,E2 -20012.819} C_VEL
LIN {X 0,Y 277.694,Z 455.883,A -85,B 0,C 180,E1 -20014.878,E2 -20014.878} C_VEL
LIN {X 0,Y 279.125,Z 458.794,A -85,B 0,C 180,E1 -20015.334,E2 -20015.334} C_VEL
LIN {X 0,Y 274.305,Z 535.421,A -85,B 0,C 180,E1 -20017.155,E2 -20017.155} C_VEL
LIN {X 0,Y 273,Z 551.423,A -85,B 0,C 180,E1 -20017.702,E2 -20017.702} C_VEL
LIN {X 0,Y 270.781,Z 566.757,A -85,B 0,C 180,E1 -20018.463,E2 -20018.463} C_VEL
LIN {X 0,Y 267.993,Z 581.291,A -85,B 0,C 180,E1 -20019.475,E2 -20019.475} C_VEL
LIN {X 0,Y 264.422,Z 595.585,A -85,B 0,C 180,E1 -20020.756,E2 -20020.756} C_VEL
LIN {X 0,Y 260.753,Z 608.479,A -85,B 0,C 180,E1 -20022.263,E2 -20022.263} C_VEL
LIN {X 0,Y 256.179,Z 621.958,A -85,B 0,C 180,E1 -20024.216,E2 -20024.216} C_VEL
LIN {X 0,Y 251.972,Z 632.909,A -85,B 0,C 180,E1 -20026.19,E2 -20026.19} C_VEL
LIN {X 0,Y 247.975,Z 642.296,A -85,B 0,C 180,E1 -20028.239,E2 -20028.239} C_VEL
LIN {X 0,Y 243.836,Z 651.418,A -85,B 0,C 180,E1 -20030.647,E2 -20030.647} C_VEL
LIN {X 0,Y 239.578,Z 660.322,A -85,B 0,C 180,E1 -20033.556,E2 -20033.556} C_VEL
LIN {X 0,Y 235.989,Z 667.556,A -85,B 0,C 180,E1 -20036.5,E2 -20036.5} C_VEL
LIN {X 0,Y 232.43,Z 674.441,A -85,B 0,C 180,E1 -20040.072,E2 -20040.072} C_VEL
LIN {X 0,Y 229.741,Z 679.672,A -85,B 0,C 180,E1 -20043.668,E2 -20043.668} C_VEL
LIN {X 0,Y 227.548,Z 683.987,A -85,B 0,C 180,E1 -20047.91,E2 -20047.91} C_VEL
LIN {X 0,Y 226.234,Z 686.482,A -85,B 0,C 180,E1 -20051.902,E2 -20051.902} C_VEL
LIN {X 0,Y 225.705,Z 687.525,A -85,B 0,C 180,E1 -20055.576,E2 -20055.576} C_VEL
LIN {X 0,Y 225.405,Z 687.414,A -85,B 0,C 180,E1 -20059.218,E2 -20059.218} C_VEL
LIN {X 0,Y 225.54,Z 686.111,A -85,B 0,C 180,E1 -20062.84,E2 -20062.84} C_VEL
LIN {X 0,Y 225.818,Z 684.896,A -85,B 0,C 180,E1 -20064.833,E2 -20064.833} C_VEL
LIN {X 0,Y 226.139,Z 681.964,A -85,B 0,C 180,E1 -20068.219,E2 -20068.219} C_VEL
LIN {X 0,Y 227.023,Z 677.678,A -85,B 0,C 180,E1 -20071.774,E2 -20071.774} C_VEL
LIN {X 0,Y 228.336,Z 672.073,A -85,B 0,C 180,E1 -20075.298,E2 -20075.298} C_VEL
LIN {X 0,Y 230.288,Z 664.983,A -85,B 0,C 180,E1 -20078.777,E2 -20078.777} C_VEL
LIN {X 0,Y 232.667,Z 657.388,A -85,B 0,C 180,E1 -20081.765,E2 -20081.765} C_VEL
LIN {X 0,Y 235.423,Z 648.28,A -85,B 0,C 180,E1 -20084.7,E2 -20084.7} C_VEL
LIN {X 0,Y 238.183,Z 639.022,A -85,B 0,C 180,E1 -20087.162,E2 -20087.162} C_VEL
LIN {X 0,Y 241.716,Z 627.029,A -85,B 0,C 180,E1 -20089.755,E2 -20089.755} C_VEL
LIN {X 0,Y 244.887,Z 614.83,A -85,B 0,C 180,E1 -20091.906,E2 -20091.906} C_VEL
LIN {X 0,Y 248.078,Z 601.389,A -85,B 0,C 180,E1 -20093.81,E2 -20093.81} C_VEL
LIN {X 0,Y 250.764,Z 588.201,A -85,B 0,C 180,E1 -20095.303,E2 -20095.303} C_VEL
LIN {X 0,Y 253.191,Z 573.711,A -85,B 0,C 180,E1 -20096.59,E2 -20096.59} C_VEL
LIN {X 0,Y 255.326,Z 557.826,A -85,B 0,C 180,E1 -20097.622,E2 -20097.622} C_VEL
LIN {X 0,Y 256.671,Z 542.815,A -85,B 0,C 180,E1 -20098.297,E2 -20098.297} C_VEL
LIN {X 0,Y 261.42,Z 445.093,A -85,B 0,C 180,E1 -20100.879,E2 -20100.879} C_VEL
LIN {X 0,Y 255.167,Z 430.404,A -85,B 0,C 180,E1 -20102.462,E2 -20102.462} C_VEL
LIN {X 0,Y 246.661,Z 415.105,A -85,B 0,C 180,E1 -20104.63,E2 -20104.63} C_VEL
LIN {X 0,Y 238.532,Z 402.169,A -85,B 0,C 180,E1 -20106.844,E2 -20106.844} C_VEL
LIN {X 0,Y 233.035,Z 394.156,A -85,B 0,C 180,E1 -20108.447,E2 -20108.447} C_VEL
LIN {X 0,Y 230.614,Z 390.509,A -85,B 0,C 180,E1 -20109.197,E2 -20109.197} C_VEL
LIN {X 0,Y 228.66,Z 388.306,A -85,B 0,C 180,E1 -20109.789,E2 -20109.789} C_VEL
LIN {X 0,Y 227.814,Z 385.714,A -85,B 0,C 180,E1 -20110.159,E2 -20110.159} C_VEL
LIN {X 0,Y 227.822,Z 385.713,A -85,B 0,C 180,E1 -20114.803,E2 -20114.803} C_VEL
LIN {X 0,Y 227.801,Z 385.732,A -85,B 0,C 180,E1 -20119.617,E2 -20119.617} C_VEL
LIN {X 0,Y 227.865,Z 385.726,A -85,B 0,C 180,E1 -20124.124,E2 -20124.124} C_VEL
LIN {X 0,Y 227.859,Z 385.73,A -85,B 0,C 180,E1 -20128.375,E2 -20128.375} C_VEL
LIN {X 0,Y 227.838,Z 385.669,A -85,B 0,C 180,E1 -20132.438,E2 -20132.438} C_VEL
LIN {X 0,Y 227.861,Z 385.687,A -85,B 0,C 180,E1 -20136.361,E2 -20136.361} C_VEL
LIN {X 0,Y 227.925,Z 385.716,A -85,B 0,C 180,E1 -20140.172,E2 -20140.172} C_VEL
LIN {X 0,Y 228.027,Z 385.693,A -85,B 0,C 180,E1 -20143.895,E2 -20143.895} C_VEL
LIN {X 0,Y 228.06,Z 385.683,A -85,B 0,C 180,E1 -20147.542,E2 -20147.542} C_VEL
LIN {X 0,Y 228.26,Z 385.672,A -85,B 0,C 180,E1 -20151.143,E2 -20151.143} C_VEL
LIN {X 0,Y 228.308,Z 385.663,A -85,B 0,C 180,E1 -20152.926,E2 -20152.926} C_VEL
LIN {X 0,Y 228.539,Z 385.641,A -85,B 0,C 180,E1 -20158.237,E2 -20158.237} C_VEL
LIN {X 0,Y 228.542,Z 385.62,A -85,B 0,C 180,E1 -20161.761,E2 -20161.761} C_VEL
LIN {X 0,Y 228.303,Z 385.658,A -85,B 0,C 180,E1 -20167.072,E2 -20167.072} C_VEL
LIN {X 0,Y 228.194,Z 385.681,A -85,B 0,C 180,E1 -20170.095,E2 -20170.095} C_VEL
LIN {X 0,Y 227.408,Z 385.779,A -85,B 0,C 180,E1 -20171.566,E2 -20171.566} C_VEL
LIN {X 0,Y 224.482,Z 386.139,A -85,B 0,C 180,E1 -20173.965,E2 -20173.965} C_VEL
LIN {X 0,Y 222.05,Z 386.445,A -85,B 0,C 180,E1 -20175.922,E2 -20175.922} C_VEL
LIN {X 0,Y 220.997,Z 386.566,A -85,B 0,C 180,E1 -20177.442,E2 -20177.442} C_VEL
LIN {X 0,Y 220.901,Z 386.577,A -85,B 0,C 180,E1 -20177.958,E2 -20177.958} C_VEL
LIN {X 0,Y 220.87,Z 386.584,A -85,B 0,C 180,E1 -20182.665,E2 -20182.665} C_VEL
LIN {X 0,Y 220.865,Z 386.59,A -85,B 0,C 180,E1 -20187.004,E2 -20187.004} C_VEL
LIN {X 0,Y 220.818,Z 386.6,A -85,B 0,C 180,E1 -20190.758,E2 -20190.758} C_VEL
LIN {X 0,Y 220.791,Z 386.605,A -85,B 0,C 180,E1 -20194.956,E2 -20194.956} C_VEL
LIN {X 0,Y 220.824,Z 386.679,A -85,B 0,C 180,E1 -20197.206,E2 -20197.206} C_VEL
LIN {X 0,Y 221.058,Z 387.818,A -85,B 0,C 180,E1 -20197.733,E2 -20197.733} C_VEL
LIN {X 0,Y 222.453,Z 390.335,A -85,B 0,C 180,E1 -20198.243,E2 -20198.243} C_VEL
LIN {X 0,Y 225.123,Z 394.098,A -85,B 0,C 180,E1 -20199.142,E2 -20199.142} C_VEL
LIN {X 0,Y 231.688,Z 404.925,A -85,B 0,C 180,E1 -20201.281,E2 -20201.281} C_VEL
LIN {X 0,Y 238.43,Z 417.167,A -85,B 0,C 180,E1 -20203.332,E2 -20203.332} C_VEL
LIN {X 0,Y 245.328,Z 430.936,A -85,B 0,C 180,E1 -20205.3,E2 -20205.3} C_VEL
LIN {X 0,Y 251.696,Z 445.962,A -85,B 0,C 180,E1 -20207.061,E2 -20207.061} C_VEL
LIN {X 0,Y 255.417,Z 455.561,A -85,B 0,C 180,E1 -20208.061,E2 -20208.061} C_VEL
LIN {X 0,Y 250.509,Z 554.693,A -85,B 0,C 180,E1 -20210.729,E2 -20210.729} C_VEL
LIN {X 0,Y 248.947,Z 570.362,A -85,B 0,C 180,E1 -20211.411,E2 -20211.411} C_VEL
LIN {X 0,Y 246.677,Z 585.392,A -85,B 0,C 180,E1 -20212.355,E2 -20212.355} C_VEL
LIN {X 0,Y 244.274,Z 598.577,A -85,B 0,C 180,E1 -20213.485,E2 -20213.485} C_VEL
LIN {X 0,Y 241.447,Z 611.661,A -85,B 0,C 180,E1 -20214.909,E2 -20214.909} C_VEL
LIN {X 0,Y 238.269,Z 624.613,A -85,B 0,C 180,E1 -20216.676,E2 -20216.676} C_VEL
LIN {X 0,Y 234.987,Z 636.582,A -85,B 0,C 180,E1 -20218.691,E2 -20218.691} C_VEL
LIN {X 0,Y 231.649,Z 647.659,A -85,B 0,C 180,E1 -20220.96,E2 -20220.96} C_VEL
LIN {X 0,Y 228.657,Z 657.896,A -85,B 0,C 180,E1 -20223.533,E2 -20223.533} C_VEL
LIN {X 0,Y 225.548,Z 667.86,A -85,B 0,C 180,E1 -20226.591,E2 -20226.591} C_VEL
LIN {X 0,Y 223.066,Z 676.159,A -85,B 0,C 180,E1 -20229.722,E2 -20229.722} C_VEL
LIN {X 0,Y 220.93,Z 683.88,A -85,B 0,C 180,E1 -20233.363,E2 -20233.363} C_VEL
LIN {X 0,Y 219.514,Z 690.01,A -85,B 0,C 180,E1 -20237.049,E2 -20237.049} C_VEL
LIN {X 0,Y 218.815,Z 694.711,A -85,B 0,C 180,E1 -20240.759,E2 -20240.759} C_VEL
LIN {X 0,Y 218.56,Z 698.076,A -85,B 0,C 180,E1 -20244.464,E2 -20244.464} C_VEL
LIN {X 0,Y 218.606,Z 700.205,A -85,B 0,C 180,E1 -20248.158,E2 -20248.158} C_VEL
LIN {X 0,Y 218.677,Z 700.826,A -85,B 0,C 180,E1 -20250,E2 -20250} C_VEL
LIN {X 0,Y 218.496,Z 701.194,A -85,B 0,C 180,E1 -20253.688,E2 -20253.688} C_VEL
LIN {X 0,Y 218.574,Z 700.432,A -85,B 0,C 180,E1 -20257.39,E2 -20257.39} C_VEL
LIN {X 0,Y 219.158,Z 698.482,A -85,B 0,C 180,E1 -20261.093,E2 -20261.093} C_VEL
LIN {X 0,Y 220.449,Z 695.373,A -85,B 0,C 180,E1 -20264.776,E2 -20264.776} C_VEL
LIN {X 0,Y 222.493,Z 690.769,A -85,B 0,C 180,E1 -20268.628,E2 -20268.628} C_VEL
LIN {X 0,Y 225.211,Z 685.409,A -85,B 0,C 180,E1 -20271.992,E2 -20271.992} C_VEL
LIN {X 0,Y 228.801,Z 678.301,A -85,B 0,C 180,E1 -20275.47,E2 -20275.47} C_VEL
LIN {X 0,Y 232.721,Z 670.74,A -85,B 0,C 180,E1 -20278.401,E2 -20278.401} C_VEL
LIN {X 0,Y 237.061,Z 661.684,A -85,B 0,C 180,E1 -20281.253,E2 -20281.253} C_VEL
LIN {X 0,Y 242.111,Z 650.776,A -85,B 0,C 180,E1 -20283.972,E2 -20283.972} C_VEL
LIN {X 0,Y 246.909,Z 639.608,A -85,B 0,C 180,E1 -20286.202,E2 -20286.202} C_VEL
LIN {X 0,Y 251.951,Z 626.67,A -85,B 0,C 180,E1 -20288.251,E2 -20288.251} C_VEL
LIN {X 0,Y 256.018,Z 614.364,A -85,B 0,C 180,E1 -20289.84,E2 -20289.84} C_VEL
LIN {X 0,Y 259.98,Z 600.736,A -85,B 0,C 180,E1 -20291.218,E2 -20291.218} C_VEL
LIN {X 0,Y 263.22,Z 587.425,A -85,B 0,C 180,E1 -20292.261,E2 -20292.261} C_VEL
LIN {X 0,Y 266.085,Z 572.863,A -85,B 0,C 180,E1 -20293.112,E2 -20293.112} C_VEL
LIN {X 0,Y 268.177,Z 558.039,A -85,B 0,C 180,E1 -20293.725,E2 -20293.725} C_VEL
LIN {X 0,Y 269.676,Z 538.603,A -85,B 0,C 180,E1 -20294.262,E2 -20294.262} C_VEL
LIN {X 0,Y 273.883,Z 469.413,A -85,B 0,C 180,E1 -20295.989,E2 -20295.989} C_VEL
LIN {X 0,Y 268.098,Z 456.746,A -85,B 0,C 180,E1 -20298.026,E2 -20298.026} C_VEL
LIN {X 0,Y 262.016,Z 444.868,A -85,B 0,C 180,E1 -20300.317,E2 -20300.317} C_VEL
LIN {X 0,Y 255.373,Z 433.192,A -85,B 0,C 180,E1 -20303.048,E2 -20303.048} C_VEL
LIN {X 0,Y 248.845,Z 422.684,A -85,B 0,C 180,E1 -20306.066,E2 -20306.066} C_VEL
LIN {X 0,Y 244.104,Z 415.76,A -85,B 0,C 180,E1 -20308.516,E2 -20308.516} C_VEL
LIN {X 0,Y 240.696,Z 410.966,A -85,B 0,C 180,E1 -20310.467,E2 -20310.467} C_VEL
LIN {X 0,Y 236.535,Z 405.244,A -85,B 0,C 180,E1 -20313.153,E2 -20313.153} C_VEL
LIN {X 0,Y 233.774,Z 402.248,A -85,B 0,C 180,E1 -20315.11,E2 -20315.11} C_VEL
LIN {X 0,Y 231.812,Z 399.266,A -85,B 0,C 180,E1 -20316.73,E2 -20316.73} C_VEL
LIN {X 0,Y 231.306,Z 398.434,A -85,B 0,C 180,E1 -20317.181,E2 -20317.181} C_VEL
LIN {X 0,Y 228.416,Z 396.414,A -85,B 0,C 180,E1 -20319.749,E2 -20319.749} C_VEL
LIN {X 0,Y 226.918,Z 393.866,A -85,B 0,C 180,E1 -20321.491,E2 -20321.491} C_VEL
LIN {X 0,Y 226.476,Z 392.633,A -85,B 0,C 180,E1 -20322.118,E2 -20322.118} C_VEL
LIN {X 0,Y 223.039,Z 390.732,A -85,B 0,C 180,E1 -20327.027,E2 -20327.027} C_VEL
LIN {X 0,Y 221.304,Z 386.977,A -85,B 0,C 180,E1 -20333.161,E2 -20333.161} C_VEL
LIN {X 0,Y 221.512,Z 386.552,A -85,B 0,C 180,E1 -20338.183,E2 -20338.183} C_VEL
LIN {X 0,Y 223.635,Z 391.154,A -85,B 0,C 180,E1 -20344.507,E2 -20344.507} C_VEL
LIN {X 0,Y 226.839,Z 392.719,A -85,B 0,C 180,E1 -20348.744,E2 -20348.744} C_VEL
LIN {X 0,Y 227.954,Z 395.518,A -85,B 0,C 180,E1 -20350.191,E2 -20350.191} C_VEL
LIN {X 0,Y 230.163,Z 397.786,A -85,B 0,C 180,E1 -20352.343,E2 -20352.343} C_VEL
LIN {X 0,Y 231.753,Z 398.689,A -85,B 0,C 180,E1 -20353.641,E2 -20353.641} C_VEL
LIN {X 0,Y 233.395,Z 401.645,A -85,B 0,C 180,E1 -20355.054,E2 -20355.054} C_VEL
LIN {X 0,Y 236.349,Z 404.323,A -85,B 0,C 180,E1 -20357.133,E2 -20357.133} C_VEL
LIN {X 0,Y 238.781,Z 407.906,A -85,B 0,C 180,E1 -20358.78,E2 -20358.78} C_VEL
LIN {X 0,Y 240.658,Z 409.826,A -85,B 0,C 180,E1 -20359.902,E2 -20359.902} C_VEL
LIN {X 0,Y 243.235,Z 413.327,A -85,B 0,C 180,E1 -20361.395,E2 -20361.395} C_VEL
LIN {X 0,Y 244.837,Z 415.126,A -85,B 0,C 180,E1 -20362.244,E2 -20362.244} C_VEL
LIN {X 0,Y 247.757,Z 418.836,A -85,B 0,C 180,E1 -20363.732,E2 -20363.732} C_VEL
LIN {X 0,Y 252.954,Z 425.98,A -85,B 0,C 180,E1 -20366.173,E2 -20366.173} C_VEL
LIN {X 0,Y 257.78,Z 432.804,A -85,B 0,C 180,E1 -20368.22,E2 -20368.22} C_VEL
LIN {X 0,Y 264.071,Z 442.308,A -85,B 0,C 180,E1 -20370.653,E2 -20370.653} C_VEL
LIN {X 0,Y 269.009,Z 450.858,A -85,B 0,C 180,E1 -20372.439,E2 -20372.439} C_VEL
LIN {X 0,Y 274.306,Z 461.567,A -85,B 0,C 180,E1 -20374.269,E2 -20374.269} C_VEL
LIN {X 0,Y 269.848,Z 531.003,A -85,B 0,C 180,E1 -20375.946,E2 -20375.946} C_VEL
LIN {X 0,Y 268.473,Z 548.453,A -85,B 0,C 180,E1 -20376.472,E2 -20376.472} C_VEL
LIN {X 0,Y 266.447,Z 563.217,A -85,B 0,C 180,E1 -20377.149,E2 -20377.149} C_VEL
LIN {X 0,Y 263.848,Z 577.497,A -85,B 0,C 180,E1 -20378.084,E2 -20378.084} C_VEL
LIN {X 0,Y 260.657,Z 590.716,A -85,B 0,C 180,E1 -20379.179,E2 -20379.179} C_VEL
LIN {X 0,Y 257.388,Z 602.539,A -85,B 0,C 180,E1 -20380.428,E2 -20380.428} C_VEL
LIN {X 0,Y 252.881,Z 616.398,A -85,B 0,C 180,E1 -20382.272,E2 -20382.272} C_VEL
LIN {X 0,Y 248.125,Z 628.857,A -85,B 0,C 180,E1 -20384.341,E2 -20384.341} C_VEL
LIN {X 0,Y 243.244,Z 640.154,A -85,B 0,C 180,E1 -20386.67,E2 -20386.67} C_VEL
LIN {X 0,Y 238.901,Z 649.671,A -85,B 0,C 180,E1 -20389.114,E2 -20389.114} C_VEL
LIN {X 0,Y 234.296,Z 658.92,A -85,B 0,C 180,E1 -20392.054,E2 -20392.054} C_VEL
LIN {X 0,Y 230.003,Z 667.075,A -85,B 0,C 180,E1 -20395.327,E2 -20395.327} C_VEL
LIN {X 0,Y 226.047,Z 674.36,A -85,B 0,C 180,E1 -20399.136,E2 -20399.136} C_VEL
LIN {X 0,Y 223.133,Z 679.667,A -85,B 0,C 180,E1 -20402.825,E2 -20402.825} C_VEL
LIN {X 0,Y 221.444,Z 682.689,A -85,B 0,C 180,E1 -20405.633,E2 -20405.633} C_VEL
LIN {X 0,Y 219.844,Z 685.619,A -85,B 0,C 180,E1 -20409.412,E2 -20409.412} C_VEL
LIN {X 0,Y 218.883,Z 687.323,A -85,B 0,C 180,E1 -20413.203,E2 -20413.203} C_VEL
LIN {X 0,Y 218.47,Z 687.851,A -85,B 0,C 180,E1 -20416.986,E2 -20416.986} C_VEL
LIN {X 0,Y 218.339,Z 687.187,A -85,B 0,C 180,E1 -20420.738,E2 -20420.738} C_VEL
LIN {X 0,Y 218.733,Z 685.081,A -85,B 0,C 180,E1 -20424.914,E2 -20424.914} C_VEL
LIN {X 0,Y 219.049,Z 682.37,A -85,B 0,C 180,E1 -20428.162,E2 -20428.162} C_VEL
LIN {X 0,Y 219.938,Z 678.156,A -85,B 0,C 180,E1 -20431.831,E2 -20431.831} C_VEL
LIN {X 0,Y 221.282,Z 672.628,A -85,B 0,C 180,E1 -20435.468,E2 -20435.468} C_VEL
LIN {X 0,Y 223.307,Z 665.621,A -85,B 0,C 180,E1 -20439.054,E2 -20439.054} C_VEL
LIN {X 0,Y 225.735,Z 658.122,A -85,B 0,C 180,E1 -20442.131,E2 -20442.131} C_VEL
LIN {X 0,Y 228.584,Z 649.117,A -85,B 0,C 180,E1 -20445.15,E2 -20445.15} C_VEL
LIN {X 0,Y 231.997,Z 638.248,A -85,B 0,C 180,E1 -20448.09,E2 -20448.09} C_VEL
LIN {X 0,Y 235.387,Z 627.079,A -85,B 0,C 180,E1 -20450.538,E2 -20450.538} C_VEL
LIN {X 0,Y 238.683,Z 614.845,A -85,B 0,C 180,E1 -20452.735,E2 -20452.735} C_VEL
LIN {X 0,Y 242.002,Z 601.346,A -85,B 0,C 180,E1 -20454.675,E2 -20454.675} C_VEL
LIN {X 0,Y 244.798,Z 588.111,A -85,B 0,C 180,E1 -20456.194,E2 -20456.194} C_VEL
LIN {X 0,Y 247.318,Z 573.529,A -85,B 0,C 180,E1 -20457.502,E2 -20457.502} C_VEL
LIN {X 0,Y 249.435,Z 558.286,A -85,B 0,C 180,E1 -20458.505,E2 -20458.505} C_VEL
LIN {X 0,Y 250.822,Z 543.373,A -85,B 0,C 180,E1 -20459.191,E2 -20459.191} C_VEL
LIN {X 0,Y 255.766,Z 447.691,A -85,B 0,C 180,E1 -20461.747,E2 -20461.747} C_VEL
LIN {X 0,Y 252.56,Z 439.496,A -85,B 0,C 180,E1 -20462.607,E2 -20462.607} C_VEL
LIN {X 0,Y 248.778,Z 431.533,A -85,B 0,C 180,E1 -20463.602,E2 -20463.602} C_VEL
LIN {X 0,Y 241.24,Z 417.995,A -85,B 0,C 180,E1 -20465.629,E2 -20465.629} C_VEL
LIN {X 0,Y 233.996,Z 406.479,A -85,B 0,C 180,E1 -20467.701,E2 -20467.701} C_VEL
LIN {X 0,Y 228.877,Z 399.023,A -85,B 0,C 180,E1 -20469.261,E2 -20469.261} C_VEL
LIN {X 0,Y 226.689,Z 395.83,A -85,B 0,C 180,E1 -20469.963,E2 -20469.963} C_VEL
LIN {X 0,Y 224.452,Z 392.766,A -85,B 0,C 180,E1 -20470.694,E2 -20470.694} C_VEL
LIN {X 0,Y 223.667,Z 391.469,A -85,B 0,C 180,E1 -20470.966,E2 -20470.966} C_VEL
LIN {X 0,Y 221.698,Z 389.382,A -85,B 0,C 180,E1 -20471.608,E2 -20471.608} C_VEL
LIN {X 0,Y 220.84,Z 387.131,A -85,B 0,C 180,E1 -20471.958,E2 -20471.958} C_VEL
LIN {X 0,Y 220.75,Z 386.601,A -85,B 0,C 180,E1 -20472.078,E2 -20472.078} C_VEL
LIN {X 0,Y 220.761,Z 386.587,A -85,B 0,C 180,E1 -20475.541,E2 -20475.541} C_VEL
LIN {X 0,Y 220.783,Z 386.599,A -85,B 0,C 180,E1 -20480.457,E2 -20480.457} C_VEL
LIN {X 0,Y 220.828,Z 386.602,A -85,B 0,C 180,E1 -20482.792,E2 -20482.792} C_VEL
LIN {X 0,Y 220.815,Z 386.601,A -85,B 0,C 180,E1 -20487.242,E2 -20487.242} C_VEL
LIN {X 0,Y 220.797,Z 386.56,A -85,B 0,C 180,E1 -20491.48,E2 -20491.48} C_VEL
LIN {X 0,Y 220.8,Z 386.55,A -85,B 0,C 180,E1 -20495.556,E2 -20495.556} C_VEL
LIN {X 0,Y 220.878,Z 386.598,A -85,B 0,C 180,E1 -20499.512,E2 -20499.512} C_VEL
LIN {X 0,Y 220.982,Z 386.565,A -85,B 0,C 180,E1 -20503.367,E2 -20503.367} C_VEL
LIN {X 0,Y 220.999,Z 386.566,A -85,B 0,C 180,E1 -20507.137,E2 -20507.137} C_VEL
LIN {X 0,Y 221.2,Z 386.551,A -85,B 0,C 180,E1 -20510.858,E2 -20510.858} C_VEL
LIN {X 0,Y 221.245,Z 386.546,A -85,B 0,C 180,E1 -20512.699,E2 -20512.699} C_VEL
LIN {X 0,Y 221.472,Z 386.522,A -85,B 0,C 180,E1 -20518.181,E2 -20518.181} C_VEL
LIN {X 0,Y 221.475,Z 386.499,A -85,B 0,C 180,E1 -20521.818,E2 -20521.818} C_VEL
LIN {X 0,Y 221.241,Z 386.536,A -85,B 0,C 180,E1 -20527.299,E2 -20527.299} C_VEL
LIN {X 0,Y 221.061,Z 386.571,A -85,B 0,C 180,E1 -20530.996,E2 -20530.996} C_VEL
LIN {X 0,Y 220.976,Z 386.575,A -85,B 0,C 180,E1 -20536.632,E2 -20536.632} C_VEL
LIN {X 0,Y 220.901,Z 386.577,A -85,B 0,C 180,E1 -20537.958,E2 -20537.958} C_VEL
LIN {X 0,Y 220.201,Z 386.675,A -85,B 0,C 180,E1 -20539.48,E2 -20539.48} C_VEL
LIN {X 0,Y 217.321,Z 387.029,A -85,B 0,C 180,E1 -20541.964,E2 -20541.964} C_VEL
LIN {X 0,Y 214.886,Z 387.339,A -85,B 0,C 180,E1 -20543.993,E2 -20543.993} C_VEL
LIN {X 0,Y 213.838,Z 387.465,A -85,B 0,C 180,E1 -20545.569,E2 -20545.569} C_VEL
LIN {X 0,Y 213.751,Z 387.474,A -85,B 0,C 180,E1 -20546.103,E2 -20546.103} C_VEL
LIN {X 0,Y 213.768,Z 387.482,A -85,B 0,C 180,E1 -20551.262,E2 -20551.262} C_VEL
LIN {X 0,Y 213.757,Z 387.493,A -85,B 0,C 180,E1 -20555.521,E2 -20555.521} C_VEL
LIN {X 0,Y 214.668,Z 390.152,A -85,B 0,C 180,E1 -20555.943,E2 -20555.943} C_VEL
LIN {X 0,Y 216.712,Z 392.381,A -85,B 0,C 180,E1 -20556.682,E2 -20556.682} C_VEL
LIN {X 0,Y 217.364,Z 393.257,A -85,B 0,C 180,E1 -20556.92,E2 -20556.92} C_VEL
LIN {X 0,Y 221.538,Z 399.778,A -85,B 0,C 180,E1 -20558.431,E2 -20558.431} C_VEL
LIN {X 0,Y 225.834,Z 406.754,A -85,B 0,C 180,E1 -20559.899,E2 -20559.899} C_VEL
LIN {X 0,Y 231.909,Z 417.517,A -85,B 0,C 180,E1 -20561.867,E2 -20561.867} C_VEL
LIN {X 0,Y 240.044,Z 433.803,A -85,B 0,C 180,E1 -20564.336,E2 -20564.336} C_VEL
LIN {X 0,Y 246.475,Z 449.004,A -85,B 0,C 180,E1 -20566.199,E2 -20566.199} C_VEL
LIN {X 0,Y 249.727,Z 457.519,A -85,B 0,C 180,E1 -20567.12,E2 -20567.12} C_VEL
LIN {X 0,Y 244.678,Z 555.423,A -85,B 0,C 180,E1 -20569.806,E2 -20569.806} C_VEL
LIN {X 0,Y 242.954,Z 571.521,A -85,B 0,C 180,E1 -20570.543,E2 -20570.543} C_VEL
LIN {X 0,Y 240.613,Z 586.203,A -85,B 0,C 180,E1 -20571.5,E2 -20571.5} C_VEL
LIN {X 0,Y 238.025,Z 599.81,A -85,B 0,C 180,E1 -20572.709,E2 -20572.709} C_VEL
LIN {X 0,Y 234.844,Z 613.721,A -85,B 0,C 180,E1 -20574.298,E2 -20574.298} C_VEL
LIN {X 0,Y 231.205,Z 627.551,A -85,B 0,C 180,E1 -20576.306,E2 -20576.306} C_VEL
LIN {X 0,Y 227.571,Z 640.066,A -85,B 0,C 180,E1 -20578.591,E2 -20578.591} C_VEL
LIN {X 0,Y 223.724,Z 652.293,A -85,B 0,C 180,E1 -20581.376,E2 -20581.376} C_VEL
LIN {X 0,Y 220.777,Z 661.78,A -85,B 0,C 180,E1 -20584.042,E2 -20584.042} C_VEL
LIN {X 0,Y 217.737,Z 671.045,A -85,B 0,C 180,E1 -20587.211,E2 -20587.211} C_VEL
LIN {X 0,Y 215.43,Z 678.734,A -85,B 0,C 180,E1 -20590.465,E2 -20590.465} C_VEL
LIN {X 0,Y 213.611,Z 685.071,A -85,B 0,C 180,E1 -20593.76,E2 -20593.76} C_VEL
LIN {X 0,Y 212.272,Z 690.88,A -85,B 0,C 180,E1 -20597.572,E2 -20597.572} C_VEL
LIN {X 0,Y 211.762,Z 694.341,A -85,B 0,C 180,E1 -20600.448,E2 -20600.448} C_VEL
LIN {X 0,Y 211.477,Z 697.754,A -85,B 0,C 180,E1 -20604.278,E2 -20604.278} C_VEL
LIN {X 0,Y 211.502,Z 699.93,A -85,B 0,C 180,E1 -20608.096,E2 -20608.096} C_VEL
LIN {X 0,Y 211.592,Z 700.574,A -85,B 0,C 180,E1 -20610,E2 -20610} C_VEL
LIN {X 0,Y 211.394,Z 700.985,A -85,B 0,C 180,E1 -20613.812,E2 -20613.812} C_VEL
LIN {X 0,Y 211.504,Z 700.255,A -85,B 0,C 180,E1 -20617.638,E2 -20617.638} C_VEL
LIN {X 0,Y 212.138,Z 698.34,A -85,B 0,C 180,E1 -20621.465,E2 -20621.465} C_VEL
LIN {X 0,Y 213.539,Z 695.28,A -85,B 0,C 180,E1 -20625.266,E2 -20625.266} C_VEL
LIN {X 0,Y 215.587,Z 691.009,A -85,B 0,C 180,E1 -20629.026,E2 -20629.026} C_VEL
LIN {X 0,Y 218.592,Z 685.422,A -85,B 0,C 180,E1 -20632.694,E2 -20632.694} C_VEL
LIN {X 0,Y 222.385,Z 678.372,A -85,B 0,C 180,E1 -20636.26,E2 -20636.26} C_VEL
LIN {X 0,Y 226.438,Z 670.875,A -85,B 0,C 180,E1 -20639.264,E2 -20639.264} C_VEL
LIN {X 0,Y 231.002,Z 661.87,A -85,B 0,C 180,E1 -20642.169,E2 -20642.169} C_VEL
LIN {X 0,Y 236.254,Z 651.061,A -85,B 0,C 180,E1 -20644.935,E2 -20644.935} C_VEL
LIN {X 0,Y 241.67,Z 638.95,A -85,B 0,C 180,E1 -20647.378,E2 -20647.378} C_VEL
LIN {X 0,Y 246.404,Z 627.247,A -85,B 0,C 180,E1 -20649.261,E2 -20649.261} C_VEL
LIN {X 0,Y 250.298,Z 615.972,A -85,B 0,C 180,E1 -20650.755,E2 -20650.755} C_VEL
LIN {X 0,Y 254.243,Z 603.303,A -85,B 0,C 180,E1 -20652.093,E2 -20652.093} C_VEL
LIN {X 0,Y 257.53,Z 590.768,A -85,B 0,C 180,E1 -20653.154,E2 -20653.154} C_VEL
LIN {X 0,Y 260.734,Z 575.942,A -85,B 0,C 180,E1 -20654.088,E2 -20654.088} C_VEL
LIN {X 0,Y 263.159,Z 560.49,A -85,B 0,C 180,E1 -20654.779,E2 -20654.779} C_VEL
LIN {X 0,Y 264.631,Z 544.268,A -85,B 0,C 180,E1 -20655.269,E2 -20655.269} C_VEL
LIN {X 0,Y 269.217,Z 472.087,A -85,B 0,C 180,E1 -20657.075,E2 -20657.075} C_VEL
LIN {X 0,Y 263.878,Z 460.301,A -85,B 0,C 180,E1 -20659.06,E2 -20659.06} C_VEL
LIN {X 0,Y 257.532,Z 447.761,A -85,B 0,C 180,E1 -20661.594,E2 -20661.594} C_VEL
LIN {X 0,Y 251.265,Z 436.853,A -85,B 0,C 180,E1 -20664.338,E2 -20664.338} C_VEL
LIN {X 0,Y 246.23,Z 428.525,A -85,B 0,C 180,E1 -20666.802,E2 -20666.802} C_VEL
LIN {X 0,Y 241.921,Z 421.969,A -85,B 0,C 180,E1 -20669.13,E2 -20669.13} C_VEL
LIN {X 0,Y 238.29,Z 416.827,A -85,B 0,C 180,E1 -20671.303,E2 -20671.303} C_VEL
LIN {X 0,Y 234.657,Z 411.639,A -85,B 0,C 180,E1 -20673.766,E2 -20673.766} C_VEL
LIN {X 0,Y 230.519,Z 406.487,A -85,B 0,C 180,E1 -20676.987,E2 -20676.987} C_VEL
LIN {X 0,Y 229.941,Z 405.294,A -85,B 0,C 180,E1 -20677.54,E2 -20677.54} C_VEL
LIN {X 0,Y 227.046,Z 403.14,A -85,B 0,C 180,E1 -20680.212,E2 -20680.212} C_VEL
LIN {X 0,Y 225.48,Z 400.346,A -85,B 0,C 180,E1 -20682.135,E2 -20682.135} C_VEL
LIN {X 0,Y 225.251,Z 399.625,A -85,B 0,C 180,E1 -20682.487,E2 -20682.487} C_VEL
LIN {X 0,Y 221.855,Z 397.454,A -85,B 0,C 180,E1 -20687.654,E2 -20687.654} C_VEL
LIN {X 0,Y 220.43,Z 394.07,A -85,B 0,C 180,E1 -20693.134,E2 -20693.134} C_VEL
LIN {X 0,Y 220.633,Z 393.824,A -85,B 0,C 180,E1 -20698.29,E2 -20698.29} C_VEL
LIN {X 0,Y 222.628,Z 398.135,A -85,B 0,C 180,E1 -20704.301,E2 -20704.301} C_VEL
LIN {X 0,Y 225.523,Z 399.685,A -85,B 0,C 180,E1 -20708.288,E2 -20708.288} C_VEL
LIN {X 0,Y 226.776,Z 402.536,A -85,B 0,C 180,E1 -20709.927,E2 -20709.927} C_VEL
LIN {X 0,Y 229.058,Z 404.747,A -85,B 0,C 180,E1 -20712.178,E2 -20712.178} C_VEL
LIN {X 0,Y 230.227,Z 405.575,A -85,B 0,C 180,E1 -20713.173,E2 -20713.173} C_VEL
LIN {X 0,Y 232.235,Z 408.788,A -85,B 0,C 180,E1 -20714.907,E2 -20714.907} C_VEL
LIN {X 0,Y 234.636,Z 411.099,A -85,B 0,C 180,E1 -20716.645,E2 -20716.645} C_VEL
LIN {X 0,Y 237.453,Z 414.936,A -85,B 0,C 180,E1 -20718.573,E2 -20718.573} C_VEL
LIN {X 0,Y 238.639,Z 416.239,A -85,B 0,C 180,E1 -20719.308,E2 -20719.308} C_VEL
LIN {X 0,Y 241.382,Z 419.914,A -85,B 0,C 180,E1 -20720.945,E2 -20720.945} C_VEL
LIN {X 0,Y 242.864,Z 421.729,A -85,B 0,C 180,E1 -20721.764,E2 -20721.764} C_VEL
LIN {X 0,Y 246.548,Z 426.661,A -85,B 0,C 180,E1 -20723.689,E2 -20723.689} C_VEL
LIN {X 0,Y 251.838,Z 433.939,A -85,B 0,C 180,E1 -20726.186,E2 -20726.186} C_VEL
LIN {X 0,Y 259.076,Z 444.801,A -85,B 0,C 180,E1 -20729.229,E2 -20729.229} C_VEL
LIN {X 0,Y 264.522,Z 454.085,A -85,B 0,C 180,E1 -20731.316,E2 -20731.316} C_VEL
LIN {X 0,Y 269.649,Z 464.395,A -85,B 0,C 180,E1 -20733.185,E2 -20733.185} C_VEL
LIN {X 0,Y 264.289,Z 543.626,A -85,B 0,C 180,E1 -20735.144,E2 -20735.144} C_VEL
LIN {X 0,Y 262.406,Z 559.35,A -85,B 0,C 180,E1 -20735.804,E2 -20735.804} C_VEL
LIN {X 0,Y 259.997,Z 572.834,A -85,B 0,C 180,E1 -20736.595,E2 -20736.595} C_VEL
LIN {X 0,Y 256.656,Z 587.54,A -85,B 0,C 180,E1 -20737.75,E2 -20737.75} C_VEL
LIN {X 0,Y 253.122,Z 599.873,A -85,B 0,C 180,E1 -20738.974,E2 -20738.974} C_VEL
LIN {X 0,Y 249.023,Z 612.704,A -85,B 0,C 180,E1 -20740.609,E2 -20740.609} C_VEL
LIN {X 0,Y 244.327,Z 624.974,A -85,B 0,C 180,E1 -20742.515,E2 -20742.515} C_VEL
LIN {X 0,Y 239.381,Z 636.648,A -85,B 0,C 180,E1 -20744.8,E2 -20744.8} C_VEL
LIN {X 0,Y 234.844,Z 646.226,A -85,B 0,C 180,E1 -20747.092,E2 -20747.092} C_VEL
LIN {X 0,Y 229.852,Z 656.11,A -85,B 0,C 180,E1 -20750.051,E2 -20750.051} C_VEL
LIN {X 0,Y 225.438,Z 664.281,A -85,B 0,C 180,E1 -20753.122,E2 -20753.122} C_VEL
LIN {X 0,Y 221.631,Z 671.022,A -85,B 0,C 180,E1 -20756.294,E2 -20756.294} C_VEL
LIN {X 0,Y 217.968,Z 677.283,A -85,B 0,C 180,E1 -20760.122,E2 -20760.122} C_VEL
LIN {X 0,Y 215.912,Z 680.74,A -85,B 0,C 180,E1 -20762.89,E2 -20762.89} C_VEL
LIN {X 0,Y 213.668,Z 684.609,A -85,B 0,C 180,E1 -20767.072,E2 -20767.072} C_VEL
LIN {X 0,Y 212.332,Z 686.76,A -85,B 0,C 180,E1 -20770.671,E2 -20770.671} C_VEL
LIN {X 0,Y 211.636,Z 687.937,A -85,B 0,C 180,E1 -20774.594,E2 -20774.594} C_VEL
LIN {X 0,Y 211.229,Z 687.913,A -85,B 0,C 180,E1 -20778.485,E2 -20778.485} C_VEL
LIN {X 0,Y 211.314,Z 686.721,A -85,B 0,C 180,E1 -20782.355,E2 -20782.355} C_VEL
LIN {X 0,Y 211.651,Z 685.27,A -85,B 0,C 180,E1 -20784.994,E2 -20784.994} C_VEL
LIN {X 0,Y 211.96,Z 682.775,A -85,B 0,C 180,E1 -20788.1,E2 -20788.1} C_VEL
LIN {X 0,Y 212.84,Z 678.635,A -85,B 0,C 180,E1 -20791.892,E2 -20791.892} C_VEL
LIN {X 0,Y 214.232,Z 673.182,A -85,B 0,C 180,E1 -20795.648,E2 -20795.648} C_VEL
LIN {X 0,Y 216.333,Z 666.256,A -85,B 0,C 180,E1 -20799.348,E2 -20799.348} C_VEL
LIN {X 0,Y 218.815,Z 658.84,A -85,B 0,C 180,E1 -20802.521,E2 -20802.521} C_VEL
LIN {X 0,Y 221.76,Z 649.91,A -85,B 0,C 180,E1 -20805.628,E2 -20805.628} C_VEL
LIN {X 0,Y 225.289,Z 639.181,A -85,B 0,C 180,E1 -20808.648,E2 -20808.648} C_VEL
LIN {X 0,Y 229.091,Z 627.112,A -85,B 0,C 180,E1 -20811.365,E2 -20811.365} C_VEL
LIN {X 0,Y 232.537,Z 614.84,A -85,B 0,C 180,E1 -20813.607,E2 -20813.607} C_VEL
LIN {X 0,Y 235.984,Z 601.287,A -85,B 0,C 180,E1 -20815.584,E2 -20815.584} C_VEL
LIN {X 0,Y 238.895,Z 588,A -85,B 0,C 180,E1 -20817.129,E2 -20817.129} C_VEL
LIN {X 0,Y 241.509,Z 573.319,A -85,B 0,C 180,E1 -20818.459,E2 -20818.459} C_VEL
LIN {X 0,Y 243.688,Z 557.892,A -85,B 0,C 180,E1 -20819.478,E2 -20819.478} C_VEL
LIN {X 0,Y 245.128,Z 542.697,A -85,B 0,C 180,E1 -20820.175,E2 -20820.175} C_VEL
LIN {X 0,Y 250.076,Z 449.345,A -85,B 0,C 180,E1 -20822.706,E2 -20822.706} C_VEL
LIN {X 0,Y 244.894,Z 437.224,A -85,B 0,C 180,E1 -20824.144,E2 -20824.144} C_VEL
LIN {X 0,Y 236.628,Z 422.232,A -85,B 0,C 180,E1 -20826.455,E2 -20826.455} C_VEL
LIN {X 0,Y 228.366,Z 408.978,A -85,B 0,C 180,E1 -20828.954,E2 -20828.954} C_VEL
LIN {X 0,Y 222.752,Z 400.911,A -85,B 0,C 180,E1 -20830.779,E2 -20830.779} C_VEL
LIN {X 0,Y 219.689,Z 396.728,A -85,B 0,C 180,E1 -20831.83,E2 -20831.83} C_VEL
LIN {X 0,Y 217.402,Z 393.47,A -85,B 0,C 180,E1 -20832.654,E2 -20832.654} C_VEL
LIN {X 0,Y 216.84,Z 392.531,A -85,B 0,C 180,E1 -20832.868,E2 -20832.868} C_VEL
LIN {X 0,Y 214.671,Z 390.284,A -85,B 0,C 180,E1 -20833.644,E2 -20833.644} C_VEL
LIN {X 0,Y 213.783,Z 387.95,A -85,B 0,C 180,E1 -20834.043,E2 -20834.043} C_VEL
LIN {X 0,Y 213.722,Z 387.476,A -85,B 0,C 180,E1 -20834.141,E2 -20834.141} C_VEL
LIN {X 0,Y 213.705,Z 387.491,A -85,B 0,C 180,E1 -20839.147,E2 -20839.147} C_VEL
LIN {X 0,Y 213.744,Z 387.487,A -85,B 0,C 180,E1 -20843.71,E2 -20843.71} C_VEL
LIN {X 0,Y 213.762,Z 387.487,A -85,B 0,C 180,E1 -20848.26,E2 -20848.26} C_VEL
LIN {X 0,Y 213.786,Z 387.415,A -85,B 0,C 180,E1 -20852.597,E2 -20852.597} C_VEL
LIN {X 0,Y 213.782,Z 387.451,A -85,B 0,C 180,E1 -20856.999,E2 -20856.999} C_VEL
LIN {X 0,Y 213.889,Z 387.445,A -85,B 0,C 180,E1 -20862.343,E2 -20862.343} C_VEL
LIN {X 0,Y 213.939,Z 387.451,A -85,B 0,C 180,E1 -20866.705,E2 -20866.705} C_VEL
LIN {X 0,Y 214.138,Z 387.426,A -85,B 0,C 180,E1 -20870.554,E2 -20870.554} C_VEL
LIN {X 0,Y 214.077,Z 387.42,A -85,B 0,C 180,E1 -20874.347,E2 -20874.347} C_VEL
LIN {X 0,Y 214.408,Z 387.402,A -85,B 0,C 180,E1 -20878.121,E2 -20878.121} C_VEL
LIN {X 0,Y 214.517,Z 387.376,A -85,B 0,C 180,E1 -20879.999,E2 -20879.999} C_VEL
LIN {X 0,Y 214.412,Z 387.379,A -85,B 0,C 180,E1 -20881.878,E2 -20881.878} C_VEL
LIN {X 0,Y 214.182,Z 387.414,A -85,B 0,C 180,E1 -20887.541,E2 -20887.541} C_VEL
LIN {X 0,Y 213.991,Z 387.447,A -85,B 0,C 180,E1 -20891.364,E2 -20891.364} C_VEL
LIN {X 0,Y 213.88,Z 387.463,A -85,B 0,C 180,E1 -20895.24,E2 -20895.24} C_VEL
LIN {X 0,Y 213.819,Z 387.465,A -85,B 0,C 180,E1 -20899.188,E2 -20899.188} C_VEL
LIN {X 0,Y 213.804,Z 387.466,A -85,B 0,C 180,E1 -20903.231,E2 -20903.231} C_VEL
LIN {X 0,Y 213.751,Z 387.474,A -85,B 0,C 180,E1 -20906.103,E2 -20906.103} C_VEL
LIN {X 0,Y 213.062,Z 387.563,A -85,B 0,C 180,E1 -20907.15,E2 -20907.15} C_VEL
LIN {X 0,Y 210.206,Z 387.923,A -85,B 0,C 180,E1 -20908.794,E2 -20908.794} C_VEL
LIN {X 0,Y 207.348,Z 388.277,A -85,B 0,C 180,E1 -20910.482,E2 -20910.482} C_VEL
LIN {X 0,Y 206.7,Z 388.361,A -85,B 0,C 180,E1 -20911.577,E2 -20911.577} C_VEL
LIN {X 0,Y 206.673,Z 388.364,A -85,B 0,C 180,E1 -20913.179,E2 -20913.179} C_VEL
LIN {X 0,Y 207.616,Z 391.071,A -85,B 0,C 180,E1 -20913.662,E2 -20913.662} C_VEL
LIN {X 0,Y 209.645,Z 393.269,A -85,B 0,C 180,E1 -20914.478,E2 -20914.478} C_VEL
LIN {X 0,Y 210.434,Z 394.032,A -85,B 0,C 180,E1 -20914.782,E2 -20914.782} C_VEL
LIN {X 0,Y 212.426,Z 397.198,A -85,B 0,C 180,E1 -20915.596,E2 -20915.596} C_VEL
LIN {X 0,Y 213.964,Z 398.984,A -85,B 0,C 180,E1 -20916.171,E2 -20916.171} C_VEL
LIN {X 0,Y 217.732,Z 404.809,A -85,B 0,C 180,E1 -20917.591,E2 -20917.591} C_VEL
LIN {X 0,Y 223.079,Z 413.743,A -85,B 0,C 180,E1 -20919.493,E2 -20919.493} C_VEL
LIN {X 0,Y 229.516,Z 425.779,A -85,B 0,C 180,E1 -20921.648,E2 -20921.648} C_VEL
LIN {X 0,Y 236.233,Z 439.839,A -85,B 0,C 180,E1 -20923.764,E2 -20923.764} C_VEL
LIN {X 0,Y 241.862,Z 453.624,A -85,B 0,C 180,E1 -20925.474,E2 -20925.474} C_VEL
LIN {X 0,Y 244.164,Z 459.912,A -85,B 0,C 180,E1 -20926.163,E2 -20926.163} C_VEL
LIN {X 0,Y 239.022,Z 554.797,A -85,B 0,C 180,E1 -20928.79,E2 -20928.79} C_VEL
LIN {X 0,Y 237.324,Z 570.243,A -85,B 0,C 180,E1 -20929.485,E2 -20929.485} C_VEL
LIN {X 0,Y 234.825,Z 585.803,A -85,B 0,C 180,E1 -20930.507,E2 -20930.507} C_VEL
LIN {X 0,Y 232.122,Z 599.539,A -85,B 0,C 180,E1 -20931.744,E2 -20931.744} C_VEL
LIN {X 0,Y 229.056,Z 612.576,A -85,B 0,C 180,E1 -20933.251,E2 -20933.251} C_VEL
LIN {X 0,Y 225.657,Z 625.279,A -85,B 0,C 180,E1 -20935.09,E2 -20935.09} C_VEL
LIN {X 0,Y 222.141,Z 637.058,A -85,B 0,C 180,E1 -20937.194,E2 -20937.194} C_VEL
LIN {X 0,Y 218.557,Z 647.985,A -85,B 0,C 180,E1 -20939.571,E2 -20939.571} C_VEL
LIN {X 0,Y 215.222,Z 658.405,A -85,B 0,C 180,E1 -20942.375,E2 -20942.375} C_VEL
LIN {X 0,Y 211.976,Z 667.956,A -85,B 0,C 180,E1 -20945.516,E2 -20945.516} C_VEL
LIN {X 0,Y 209.285,Z 676.162,A -85,B 0,C 180,E1 -20948.838,E2 -20948.838} C_VEL
LIN {X 0,Y 207.151,Z 682.948,A -85,B 0,C 180,E1 -20952.221,E2 -20952.221} C_VEL
LIN {X 0,Y 205.593,Z 689.182,A -85,B 0,C 180,E1 -20956.155,E2 -20956.155} C_VEL
LIN {X 0,Y 204.701,Z 693.967,A -85,B 0,C 180,E1 -20960.115,E2 -20960.115} C_VEL
LIN {X 0,Y 204.379,Z 697.431,A -85,B 0,C 180,E1 -20964.079,E2 -20964.079} C_VEL
LIN {X 0,Y 204.401,Z 699.654,A -85,B 0,C 180,E1 -20968.029,E2 -20968.029} C_VEL
LIN {X 0,Y 204.508,Z 700.321,A -85,B 0,C 180,E1 -20970,E2 -20970} C_VEL
LIN {X 0,Y 204.294,Z 700.777,A -85,B 0,C 180,E1 -20973.945,E2 -20973.945} C_VEL
LIN {X 0,Y 204.434,Z 700.071,A -85,B 0,C 180,E1 -20977.904,E2 -20977.904} C_VEL
LIN {X 0,Y 205.137,Z 698.201,A -85,B 0,C 180,E1 -20981.862,E2 -20981.862} C_VEL
LIN {X 0,Y 206.65,Z 695.189,A -85,B 0,C 180,E1 -20985.788,E2 -20985.788} C_VEL
LIN {X 0,Y 208.821,Z 690.968,A -85,B 0,C 180,E1 -20989.667,E2 -20989.667} C_VEL
LIN {X 0,Y 211.995,Z 685.434,A -85,B 0,C 180,E1 -20993.442,E2 -20993.442} C_VEL
LIN {X 0,Y 216.025,Z 678.442,A -85,B 0,C 180,E1 -20997.095,E2 -20997.095} C_VEL
LIN {X 0,Y 220.196,Z 670.996,A -85,B 0,C 180,E1 -21000.178,E2 -21000.178} C_VEL
LIN {X 0,Y 225.018,Z 662.047,A -85,B 0,C 180,E1 -21003.133,E2 -21003.133} C_VEL
LIN {X 0,Y 230.474,Z 651.331,A -85,B 0,C 180,E1 -21005.945,E2 -21005.945} C_VEL
LIN {X 0,Y 236.087,Z 639.349,A -85,B 0,C 180,E1 -21008.42,E2 -21008.42} C_VEL
LIN {X 0,Y 240.948,Z 627.784,A -85,B 0,C 180,E1 -21010.316,E2 -21010.316} C_VEL
LIN {X 0,Y 244.988,Z 616.595,A -85,B 0,C 180,E1 -21011.834,E2 -21011.834} C_VEL
LIN {X 0,Y 249.568,Z 602.374,A -85,B 0,C 180,E1 -21013.347,E2 -21013.347} C_VEL
LIN {X 0,Y 252.985,Z 589.639,A -85,B 0,C 180,E1 -21014.404,E2 -21014.404} C_VEL
LIN {X 0,Y 256.153,Z 575.248,A -85,B 0,C 180,E1 -21015.299,E2 -21015.299} C_VEL
LIN {X 0,Y 258.507,Z 560.691,A -85,B 0,C 180,E1 -21015.952,E2 -21015.952} C_VEL
LIN {X 0,Y 260.028,Z 544.706,A -85,B 0,C 180,E1 -21016.443,E2 -21016.443} C_VEL
LIN {X 0,Y 264.628,Z 474.813,A -85,B 0,C 180,E1 -21018.205,E2 -21018.205} C_VEL
LIN {X 0,Y 259.768,Z 463.919,A -85,B 0,C 180,E1 -21020.118,E2 -21020.118} C_VEL
LIN {X 0,Y 253.959,Z 452.309,A -85,B 0,C 180,E1 -21022.564,E2 -21022.564} C_VEL
LIN {X 0,Y 248.343,Z 442.28,A -85,B 0,C 180,E1 -21025.154,E2 -21025.154} C_VEL
LIN {X 0,Y 243.414,Z 433.941,A -85,B 0,C 180,E1 -21027.688,E2 -21027.688} C_VEL
LIN {X 0,Y 239.772,Z 428.235,A -85,B 0,C 180,E1 -21029.75,E2 -21029.75} C_VEL
LIN {X 0,Y 236.276,Z 423.102,A -85,B 0,C 180,E1 -21031.935,E2 -21031.935} C_VEL
LIN {X 0,Y 232.896,Z 418.128,A -85,B 0,C 180,E1 -21034.324,E2 -21034.324} C_VEL
LIN {X 0,Y 228.918,Z 413.042,A -85,B 0,C 180,E1 -21037.553,E2 -21037.553} C_VEL
LIN {X 0,Y 228.36,Z 412.067,A -85,B 0,C 180,E1 -21038.09,E2 -21038.09} C_VEL
LIN {X 0,Y 225.525,Z 409.632,A -85,B 0,C 180,E1 -21040.872,E2 -21040.872} C_VEL
LIN {X 0,Y 223.833,Z 406.462,A -85,B 0,C 180,E1 -21043.117,E2 -21043.117} C_VEL
LIN {X 0,Y 220.693,Z 404.213,A -85,B 0,C 180,E1 -21048.288,E2 -21048.288} C_VEL
LIN {X 0,Y 219.498,Z 401.02,A -85,B 0,C 180,E1 -21053.676,E2 -21053.676} C_VEL
LIN {X 0,Y 219.726,Z 400.94,A -85,B 0,C 180,E1 -21058.168,E2 -21058.168} C_VEL
LIN {X 0,Y 221.624,Z 405.116,A -85,B 0,C 180,E1 -21064.092,E2 -21064.092} C_VEL
LIN {X 0,Y 224.228,Z 406.598,A -85,B 0,C 180,E1 -21067.826,E2 -21067.826} C_VEL
LIN {X 0,Y 225.663,Z 409.566,A -85,B 0,C 180,E1 -21069.722,E2 -21069.722} C_VEL
LIN {X 0,Y 228.195,Z 411.879,A -85,B 0,C 180,E1 -21072.225,E2 -21072.225} C_VEL
LIN {X 0,Y 228.839,Z 412.615,A -85,B 0,C 180,E1 -21072.81,E2 -21072.81} C_VEL
LIN {X 0,Y 231.084,Z 415.879,A -85,B 0,C 180,E1 -21074.757,E2 -21074.757} C_VEL
LIN {X 0,Y 232.95,Z 417.781,A -85,B 0,C 180,E1 -21076.149,E2 -21076.149} C_VEL
LIN {X 0,Y 235.917,Z 421.732,A -85,B 0,C 180,E1 -21078.229,E2 -21078.229} C_VEL
LIN {X 0,Y 237.144,Z 423.391,A -85,B 0,C 180,E1 -21079.027,E2 -21079.027} C_VEL
LIN {X 0,Y 240.778,Z 428.15,A -85,B 0,C 180,E1 -21081.2,E2 -21081.2} C_VEL
LIN {X 0,Y 244.162,Z 432.753,A -85,B 0,C 180,E1 -21083.035,E2 -21083.035} C_VEL
LIN {X 0,Y 249.31,Z 440.03,A -85,B 0,C 180,E1 -21085.563,E2 -21085.563} C_VEL
LIN {X 0,Y 254.636,Z 448.187,A -85,B 0,C 180,E1 -21087.928,E2 -21087.928} C_VEL
LIN {X 0,Y 260.141,Z 457.336,A -85,B 0,C 180,E1 -21090.157,E2 -21090.157} C_VEL
LIN {X 0,Y 265.009,Z 467.126,A -85,B 0,C 180,E1 -21092.033,E2 -21092.033} C_VEL
LIN {X 0,Y 262.788,Z 501.154,A -85,B 0,C 180,E1 -21092.899,E2 -21092.899} C_VEL
LIN {X 0,Y 259.741,Z 543.512,A -85,B 0,C 180,E1 -21093.954,E2 -21093.954} C_VEL
LIN {X 0,Y 257.799,Z 559.377,A -85,B 0,C 180,E1 -21094.618,E2 -21094.618} C_VEL
LIN {X 0,Y 255.2,Z 573.385,A -85,B 0,C 180,E1 -21095.438,E2 -21095.438} C_VEL
LIN {X 0,Y 251.72,Z 588.148,A -85,B 0,C 180,E1 -21096.611,E2 -21096.611} C_VEL
LIN {X 0,Y 248.07,Z 600.401,A -85,B 0,C 180,E1 -21097.841,E2 -21097.841} C_VEL
LIN {X 0,Y 243.828,Z 613.176,A -85,B 0,C 180,E1 -21099.489,E2 -21099.489} C_VEL
LIN {X 0,Y 238.969,Z 625.401,A -85,B 0,C 180,E1 -21101.414,E2 -21101.414} C_VEL
LIN {X 0,Y 233.672,Z 637.358,A -85,B 0,C 180,E1 -21103.794,E2 -21103.794} C_VEL
LIN {X 0,Y 228.695,Z 647.346,A -85,B 0,C 180,E1 -21106.255,E2 -21106.255} C_VEL
LIN {X 0,Y 223.544,Z 657.072,A -85,B 0,C 180,E1 -21109.28,E2 -21109.28} C_VEL
LIN {X 0,Y 218.958,Z 665.104,A -85,B 0,C 180,E1 -21112.421,E2 -21112.421} C_VEL
LIN {X 0,Y 214.458,Z 672.543,A -85,B 0,C 180,E1 -21116.144,E2 -21116.144} C_VEL
LIN {X 0,Y 210.724,Z 678.543,A -85,B 0,C 180,E1 -21120.13,E2 -21120.13} C_VEL
LIN {X 0,Y 208.078,Z 682.761,A -85,B 0,C 180,E1 -21123.955,E2 -21123.955} C_VEL
LIN {X 0,Y 206.142,Z 685.83,A -85,B 0,C 180,E1 -21127.974,E2 -21127.974} C_VEL
LIN {X 0,Y 204.921,Z 687.67,A -85,B 0,C 180,E1 -21132.021,E2 -21132.021} C_VEL
LIN {X 0,Y 204.338,Z 688.285,A -85,B 0,C 180,E1 -21136.069,E2 -21136.069} C_VEL
LIN {X 0,Y 204.118,Z 687.731,A -85,B 0,C 180,E1 -21140.087,E2 -21140.087} C_VEL
LIN {X 0,Y 204.439,Z 686.03,A -85,B 0,C 180,E1 -21144.081,E2 -21144.081} C_VEL
LIN {X 0,Y 204.871,Z 683.177,A -85,B 0,C 180,E1 -21148.034,E2 -21148.034} C_VEL
LIN {X 0,Y 205.741,Z 679.109,A -85,B 0,C 180,E1 -21151.958,E2 -21151.958} C_VEL
LIN {X 0,Y 207.187,Z 673.73,A -85,B 0,C 180,E1 -21155.841,E2 -21155.841} C_VEL
LIN {X 0,Y 209.368,Z 666.885,A -85,B 0,C 180,E1 -21159.662,E2 -21159.662} C_VEL
LIN {X 0,Y 212.283,Z 658.354,A -85,B 0,C 180,E1 -21163.4,E2 -21163.4} C_VEL
LIN {X 0,Y 215.484,Z 649.297,A -85,B 0,C 180,E1 -21166.582,E2 -21166.582} C_VEL
LIN {X 0,Y 218.605,Z 640.07,A -85,B 0,C 180,E1 -21169.24,E2 -21169.24} C_VEL
LIN {X 0,Y 222.265,Z 629.133,A -85,B 0,C 180,E1 -21171.81,E2 -21171.81} C_VEL
LIN {X 0,Y 225.787,Z 617.21,A -85,B 0,C 180,E1 -21174.113,E2 -21174.113} C_VEL
LIN {X 0,Y 229.344,Z 604.141,A -85,B 0,C 180,E1 -21176.136,E2 -21176.136} C_VEL
LIN {X 0,Y 232.273,Z 591.426,A -85,B 0,C 180,E1 -21177.724,E2 -21177.724} C_VEL
LIN {X 0,Y 235.165,Z 576.526,A -85,B 0,C 180,E1 -21179.177,E2 -21179.177} C_VEL
LIN {X 0,Y 237.485,Z 561.451,A -85,B 0,C 180,E1 -21180.266,E2 -21180.266} C_VEL
LIN {X 0,Y 239.104,Z 546.707,A -85,B 0,C 180,E1 -21181.018,E2 -21181.018} C_VEL
LIN {X 0,Y 240.436,Z 525.548,A -85,B 0,C 180,E1 -21181.684,E2 -21181.684} C_VEL
LIN {X 0,Y 244.476,Z 451.951,A -85,B 0,C 180,E1 -21183.671,E2 -21183.671} C_VEL
LIN {X 0,Y 243.623,Z 449.244,A -85,B 0,C 180,E1 -21183.94,E2 -21183.94} C_VEL
LIN {X 0,Y 239.609,Z 440.326,A -85,B 0,C 180,E1 -21185.096,E2 -21185.096} C_VEL
LIN {X 0,Y 232.38,Z 426.996,A -85,B 0,C 180,E1 -21187.22,E2 -21187.22} C_VEL
LIN {X 0,Y 224.737,Z 414.482,A -85,B 0,C 180,E1 -21189.634,E2 -21189.634} C_VEL
LIN {X 0,Y 219.013,Z 406.195,A -85,B 0,C 180,E1 -21191.57,E2 -21191.57} C_VEL
LIN {X 0,Y 216.124,Z 402.168,A -85,B 0,C 180,E1 -21192.607,E2 -21192.607} C_VEL
LIN {X 0,Y 213.064,Z 397.93,A -85,B 0,C 180,E1 -21193.76,E2 -21193.76} C_VEL
LIN {X 0,Y 210.728,Z 394.815,A -85,B 0,C 180,E1 -21194.675,E2 -21194.675} C_VEL
LIN {X 0,Y 209.93,Z 393.46,A -85,B 0,C 180,E1 -21195.011,E2 -21195.011} C_VEL
LIN {X 0,Y 207.762,Z 391.353,A -85,B 0,C 180,E1 -21195.866,E2 -21195.866} C_VEL
LIN {X 0,Y 206.731,Z 388.766,A -85,B 0,C 180,E1 -21196.371,E2 -21196.371} C_VEL
LIN {X 0,Y 206.667,Z 388.341,A -85,B 0,C 180,E1 -21196.443,E2 -21196.443} C_VEL
LIN {X 0,Y 206.672,Z 388.354,A -85,B 0,C 180,E1 -21201.456,E2 -21201.456} C_VEL
LIN {X 0,Y 206.703,Z 388.356,A -85,B 0,C 180,E1 -21204.688,E2 -21204.688} C_VEL
LIN {X 0,Y 206.697,Z 388.36,A -85,B 0,C 180,E1 -21209.334,E2 -21209.334} C_VEL
LIN {X 0,Y 206.68,Z 388.293,A -85,B 0,C 180,E1 -21213.764,E2 -21213.764} C_VEL
LIN {X 0,Y 206.72,Z 388.35,A -85,B 0,C 180,E1 -21218.038,E2 -21218.038} C_VEL
LIN {X 0,Y 206.829,Z 388.325,A -85,B 0,C 180,E1 -21222.192,E2 -21222.192} C_VEL
LIN {X 0,Y 206.88,Z 388.336,A -85,B 0,C 180,E1 -21226.242,E2 -21226.242} C_VEL
LIN {X 0,Y 207.082,Z 388.299,A -85,B 0,C 180,E1 -21230.229,E2 -21230.229} C_VEL
LIN {X 0,Y 207.041,Z 388.298,A -85,B 0,C 180,E1 -21234.154,E2 -21234.154} C_VEL
LIN {X 0,Y 207.348,Z 388.282,A -85,B 0,C 180,E1 -21238.057,E2 -21238.057} C_VEL
LIN {X 0,Y 207.484,Z 388.251,A -85,B 0,C 180,E1 -21239.999,E2 -21239.999} C_VEL
LIN {X 0,Y 207.352,Z 388.258,A -85,B 0,C 180,E1 -21241.942,E2 -21241.942} C_VEL
LIN {X 0,Y 207.127,Z 388.292,A -85,B 0,C 180,E1 -21247.8,E2 -21247.8} C_VEL
LIN {X 0,Y 206.91,Z 388.325,A -85,B 0,C 180,E1 -21251.758,E2 -21251.758} C_VEL
LIN {X 0,Y 206.815,Z 388.344,A -85,B 0,C 180,E1 -21255.774,E2 -21255.774} C_VEL
LIN {X 0,Y 206.754,Z 388.351,A -85,B 0,C 180,E1 -21259.871,E2 -21259.871} C_VEL
LIN {X 0,Y 206.739,Z 388.354,A -85,B 0,C 180,E1 -21264.074,E2 -21264.074} C_VEL
LIN {X 0,Y 206.717,Z 388.36,A -85,B 0,C 180,E1 -21268.422,E2 -21268.422} C_VEL
LIN {X 0,Y 206.7,Z 388.361,A -85,B 0,C 180,E1 -21271.577,E2 -21271.577} C_VEL
LIN {X 0,Y 206.97,Z 389.031,A -85,B 0,C 180,E1 -21272.45,E2 -21272.45} C_VEL
LIN {X 0,Y 207.785,Z 391.247,A -85,B 0,C 180,E1 -21273.417,E2 -21273.417} C_VEL
LIN {X 0,Y 208.753,Z 394.039,A -85,B 0,C 180,E1 -21274.137,E2 -21274.137} C_VEL
LIN {X 0,Y 210.869,Z 400.916,A -85,B 0,C 180,E1 -21275.287,E2 -21275.287} C_VEL
LIN {X 0,Y 213.263,Z 408.212,A -85,B 0,C 180,E1 -21276.419,E2 -21276.419} C_VEL
LIN {X 0,Y 214.875,Z 411.423,A -85,B 0,C 180,E1 -21277.072,E2 -21277.072} C_VEL
LIN {X 0,Y 219.492,Z 419.373,A -85,B 0,C 180,E1 -21278.783,E2 -21278.783} C_VEL
LIN {X 0,Y 225.491,Z 430.886,A -85,B 0,C 180,E1 -21280.882,E2 -21280.882} C_VEL
LIN {X 0,Y 231.489,Z 443.619,A -85,B 0,C 180,E1 -21282.863,E2 -21282.863} C_VEL
LIN {X 0,Y 236.89,Z 457.055,A -85,B 0,C 180,E1 -21284.59,E2 -21284.59} C_VEL
LIN {X 0,Y 238.611,Z 461.756,A -85,B 0,C 180,E1 -21285.131,E2 -21285.131} C_VEL
LIN {X 0,Y 233.312,Z 555.378,A -85,B 0,C 180,E1 -21287.769,E2 -21287.769} C_VEL
LIN {X 0,Y 231.484,Z 571.349,A -85,B 0,C 180,E1 -21288.529,E2 -21288.529} C_VEL
LIN {X 0,Y 228.892,Z 586.539,A -85,B 0,C 180,E1 -21289.561,E2 -21289.561} C_VEL
LIN {X 0,Y 226.271,Z 599.355,A -85,B 0,C 180,E1 -21290.739,E2 -21290.739} C_VEL
LIN {X 0,Y 222.838,Z 613.396,A -85,B 0,C 180,E1 -21292.399,E2 -21292.399} C_VEL
LIN {X 0,Y 219.036,Z 626.917,A -85,B 0,C 180,E1 -21294.439,E2 -21294.439} C_VEL
LIN {X 0,Y 215.122,Z 639.469,A -85,B 0,C 180,E1 -21296.823,E2 -21296.823} C_VEL
LIN {X 0,Y 211.165,Z 650.867,A -85,B 0,C 180,E1 -21299.499,E2 -21299.499} C_VEL
LIN {X 0,Y 207.884,Z 660.462,A -85,B 0,C 180,E1 -21302.299,E2 -21302.299} C_VEL
LIN {X 0,Y 204.984,Z 668.627,A -85,B 0,C 180,E1 -21305.165,E2 -21305.165} C_VEL
LIN {X 0,Y 202.226,Z 676.671,A -85,B 0,C 180,E1 -21308.598,E2 -21308.598} C_VEL
LIN {X 0,Y 199.849,Z 684.159,A -85,B 0,C 180,E1 -21312.607,E2 -21312.607} C_VEL
LIN {X 0,Y 198.318,Z 690.079,A -85,B 0,C 180,E1 -21316.682,E2 -21316.682} C_VEL
LIN {X 0,Y 197.66,Z 693.591,A -85,B 0,C 180,E1 -21319.759,E2 -21319.759} C_VEL
LIN {X 0,Y 197.29,Z 697.106,A -85,B 0,C 180,E1 -21323.865,E2 -21323.865} C_VEL
LIN {X 0,Y 197.304,Z 699.377,A -85,B 0,C 180,E1 -21327.959,E2 -21327.959} C_VEL
LIN {X 0,Y 197.425,Z 700.068,A -85,B 0,C 180,E1 -21330,E2 -21330} C_VEL
LIN {X 0,Y 197.202,Z 700.569,A -85,B 0,C 180,E1 -21334.087,E2 -21334.087} C_VEL
LIN {X 0,Y 197.384,Z 699.885,A -85,B 0,C 180,E1 -21338.188,E2 -21338.188} C_VEL
LIN {X 0,Y 198.129,Z 698.061,A -85,B 0,C 180,E1 -21342.288,E2 -21342.288} C_VEL
LIN {X 0,Y 199.751,Z 695.096,A -85,B 0,C 180,E1 -21346.348,E2 -21346.348} C_VEL
LIN {X 0,Y 202.107,Z 690.926,A -85,B 0,C 180,E1 -21350.349,E2 -21350.349} C_VEL
LIN {X 0,Y 205.45,Z 685.45,A -85,B 0,C 180,E1 -21354.236,E2 -21354.236} C_VEL
LIN {X 0,Y 209.72,Z 678.52,A -85,B 0,C 180,E1 -21357.98,E2 -21357.98} C_VEL
LIN {X 0,Y 214.009,Z 671.13,A -85,B 0,C 180,E1 -21361.136,E2 -21361.136} C_VEL
LIN {X 0,Y 219.088,Z 662.228,A -85,B 0,C 180,E1 -21364.151,E2 -21364.151} C_VEL
LIN {X 0,Y 223.933,Z 653.212,A -85,B 0,C 180,E1 -21366.606,E2 -21366.606} C_VEL
LIN {X 0,Y 229.166,Z 642.623,A -85,B 0,C 180,E1 -21368.953,E2 -21368.953} C_VEL
LIN {X 0,Y 234.876,Z 629.953,A -85,B 0,C 180,E1 -21371.17,E2 -21371.17} C_VEL
LIN {X 0,Y 239.239,Z 618.635,A -85,B 0,C 180,E1 -21372.791,E2 -21372.791} C_VEL
LIN {X 0,Y 243.972,Z 604.943,A -85,B 0,C 180,E1 -21374.312,E2 -21374.312} C_VEL
LIN {X 0,Y 247.721,Z 591.859,A -85,B 0,C 180,E1 -21375.464,E2 -21375.464} C_VEL
LIN {X 0,Y 251.115,Z 577.515,A -85,B 0,C 180,E1 -21376.4,E2 -21376.4} C_VEL
LIN {X 0,Y 253.833,Z 561.981,A -85,B 0,C 180,E1 -21377.126,E2 -21377.126} C_VEL
LIN {X 0,Y 255.409,Z 546.872,A -85,B 0,C 180,E1 -21377.617,E2 -21377.617} C_VEL
LIN {X 0,Y 260.147,Z 477.633,A -85,B 0,C 180,E1 -21379.371,E2 -21379.371} C_VEL
LIN {X 0,Y 256.062,Z 468.288,A -85,B 0,C 180,E1 -21381.074,E2 -21381.074} C_VEL
LIN {X 0,Y 250.803,Z 457.485,A -85,B 0,C 180,E1 -21383.407,E2 -21383.407} C_VEL
LIN {X 0,Y 245.493,Z 447.742,A -85,B 0,C 180,E1 -21385.979,E2 -21385.979} C_VEL
LIN {X 0,Y 240.753,Z 439.533,A -85,B 0,C 180,E1 -21388.538,E2 -21388.538} C_VEL
LIN {X 0,Y 237.272,Z 433.947,A -85,B 0,C 180,E1 -21390.615,E2 -21390.615} C_VEL
LIN {X 0,Y 234.189,Z 429.299,A -85,B 0,C 180,E1 -21392.644,E2 -21392.644} C_VEL
LIN {X 0,Y 231.054,Z 424.484,A -85,B 0,C 180,E1 -21394.97,E2 -21394.97} C_VEL
LIN {X 0,Y 227.251,Z 419.434,A -85,B 0,C 180,E1 -21398.216,E2 -21398.216} C_VEL
LIN {X 0,Y 226.809,Z 418.77,A -85,B 0,C 180,E1 -21398.649,E2 -21398.649} C_VEL
LIN {X 0,Y 223.966,Z 416.028,A -85,B 0,C 180,E1 -21401.624,E2 -21401.624} C_VEL
LIN {X 0,Y 222.639,Z 413.401,A -85,B 0,C 180,E1 -21403.496,E2 -21403.496} C_VEL
LIN {X 0,Y 219.494,Z 410.866,A -85,B 0,C 180,E1 -21409.112,E2 -21409.112} C_VEL
LIN {X 0,Y 218.621,Z 408.064,A -85,B 0,C 180,E1 -21413.746,E2 -21413.746} C_VEL
LIN {X 0,Y 218.842,Z 408.065,A -85,B 0,C 180,E1 -21418.16,E2 -21418.16} C_VEL
LIN {X 0,Y 220.623,Z 412.092,A -85,B 0,C 180,E1 -21423.882,E2 -21423.882} C_VEL
LIN {X 0,Y 223.026,Z 413.64,A -85,B 0,C 180,E1 -21427.47,E2 -21427.47} C_VEL
LIN {X 0,Y 224.646,Z 416.744,A -85,B 0,C 180,E1 -21429.625,E2 -21429.625} C_VEL
LIN {X 0,Y 227.301,Z 419.263,A -85,B 0,C 180,E1 -21432.274,E2 -21432.274} C_VEL
LIN {X 0,Y 229.705,Z 422.729,A -85,B 0,C 180,E1 -21434.423,E2 -21434.423} C_VEL
LIN {X 0,Y 231.353,Z 424.532,A -85,B 0,C 180,E1 -21435.698,E2 -21435.698} C_VEL
LIN {X 0,Y 234.206,Z 428.347,A -85,B 0,C 180,E1 -21437.759,E2 -21437.759} C_VEL
LIN {X 0,Y 238.742,Z 434.54,A -85,B 0,C 180,E1 -21440.636,E2 -21440.636} C_VEL
LIN {X 0,Y 243.059,Z 440.582,A -85,B 0,C 180,E1 -21443.033,E2 -21443.033} C_VEL
LIN {X 0,Y 248.911,Z 449.283,A -85,B 0,C 180,E1 -21445.921,E2 -21445.921} C_VEL
LIN {X 0,Y 255.199,Z 459.58,A -85,B 0,C 180,E1 -21448.686,E2 -21448.686} C_VEL
LIN {X 0,Y 258.938,Z 466.678,A -85,B 0,C 180,E1 -21450.223,E2 -21450.223} C_VEL
LIN {X 0,Y 260.606,Z 470.193,A -85,B 0,C 180,E1 -21450.893,E2 -21450.893} C_VEL
LIN {X 0,Y 255.775,Z 537.136,A -85,B 0,C 180,E1 -21452.519,E2 -21452.519} C_VEL
LIN {X 0,Y 254.236,Z 552.815,A -85,B 0,C 180,E1 -21453.076,E2 -21453.076} C_VEL
LIN {X 0,Y 251.851,Z 567.236,A -85,B 0,C 180,E1 -21453.793,E2 -21453.793} C_VEL
LIN {X 0,Y 248.51,Z 582.645,A -85,B 0,C 180,E1 -21454.902,E2 -21454.902} C_VEL
LIN {X 0,Y 244.67,Z 596.025,A -85,B 0,C 180,E1 -21456.111,E2 -21456.111} C_VEL
LIN {X 0,Y 240.13,Z 609.926,A -85,B 0,C 180,E1 -21457.794,E2 -21457.794} C_VEL
LIN {X 0,Y 235.174,Z 622.536,A -85,B 0,C 180,E1 -21459.689,E2 -21459.689} C_VEL
LIN {X 0,Y 230.449,Z 633.069,A -85,B 0,C 180,E1 -21461.654,E2 -21461.654} C_VEL
LIN {X 0,Y 225.072,Z 643.769,A -85,B 0,C 180,E1 -21464.095,E2 -21464.095} C_VEL
LIN {X 0,Y 220.245,Z 652.792,A -85,B 0,C 180,E1 -21466.681,E2 -21466.681} C_VEL
LIN {X 0,Y 215.099,Z 661.604,A -85,B 0,C 180,E1 -21469.812,E2 -21469.812} C_VEL
LIN {X 0,Y 210.312,Z 669.347,A -85,B 0,C 180,E1 -21473.324,E2 -21473.324} C_VEL
LIN {X 0,Y 206.32,Z 675.574,A -85,B 0,C 180,E1 -21476.974,E2 -21476.974} C_VEL
LIN {X 0,Y 202.868,Z 680.739,A -85,B 0,C 180,E1 -21480.987,E2 -21480.987} C_VEL
LIN {X 0,Y 200.306,Z 684.525,A -85,B 0,C 180,E1 -21485.1,E2 -21485.1} C_VEL
LIN {X 0,Y 198.529,Z 687.039,A -85,B 0,C 180,E1 -21489.268,E2 -21489.268} C_VEL
LIN {X 0,Y 197.561,Z 688.374,A -85,B 0,C 180,E1 -21493.845,E2 -21493.845} C_VEL
LIN {X 0,Y 197.096,Z 688.39,A -85,B 0,C 180,E1 -21497.646,E2 -21497.646} C_VEL
LIN {X 0,Y 197.09,Z 687.329,A -85,B 0,C 180,E1 -21501.8,E2 -21501.8} C_VEL
LIN {X 0,Y 197.525,Z 685.119,A -85,B 0,C 180,E1 -21505.919,E2 -21505.919} C_VEL
LIN {X 0,Y 198.077,Z 681.741,A -85,B 0,C 180,E1 -21510,E2 -21510} C_VEL
LIN {X 0,Y 199.336,Z 677.097,A -85,B 0,C 180,E1 -21514.044,E2 -21514.044} C_VEL
LIN {X 0,Y 201.198,Z 671.074,A -85,B 0,C 180,E1 -21518.032,E2 -21518.032} C_VEL
LIN {X 0,Y 203.827,Z 663.51,A -85,B 0,C 180,E1 -21521.94,E2 -21521.94} C_VEL
LIN {X 0,Y 206.762,Z 655.411,A -85,B 0,C 180,E1 -21525.274,E2 -21525.274} C_VEL
LIN {X 0,Y 210.262,Z 645.711,A -85,B 0,C 180,E1 -21528.514,E2 -21528.514} C_VEL
LIN {X 0,Y 213.783,Z 635.783,A -85,B 0,C 180,E1 -21531.2,E2 -21531.2} C_VEL
LIN {X 0,Y 217.647,Z 624,A -85,B 0,C 180,E1 -21533.806,E2 -21533.806} C_VEL
LIN {X 0,Y 221.143,Z 612.262,A -85,B 0,C 180,E1 -21535.912,E2 -21535.912} C_VEL
LIN {X 0,Y 224.525,Z 599.593,A -85,B 0,C 180,E1 -21537.75,E2 -21537.75} C_VEL
LIN {X 0,Y 227.68,Z 585.765,A -85,B 0,C 180,E1 -21539.343,E2 -21539.343} C_VEL
LIN {X 0,Y 230.294,Z 571.538,A -85,B 0,C 180,E1 -21540.615,E2 -21540.615} C_VEL
LIN {X 0,Y 232.532,Z 556.101,A -85,B 0,C 180,E1 -21541.614,E2 -21541.614} C_VEL
LIN {X 0,Y 233.939,Z 540.995,A -85,B 0,C 180,E1 -21542.289,E2 -21542.289} C_VEL
LIN {X 0,Y 238.924,Z 453.399,A -85,B 0,C 180,E1 -21544.726,E2 -21544.726} C_VEL
LIN {X 0,Y 234.956,Z 444.467,A -85,B 0,C 180,E1 -21545.924,E2 -21545.924} C_VEL
LIN {X 0,Y 228.225,Z 431.839,A -85,B 0,C 180,E1 -21547.997,E2 -21547.997} C_VEL
LIN {X 0,Y 220.819,Z 419.516,A -85,B 0,C 180,E1 -21550.443,E2 -21550.443} C_VEL
LIN {X 0,Y 215.308,Z 411.425,A -85,B 0,C 180,E1 -21552.394,E2 -21552.394} C_VEL
LIN {X 0,Y 211.818,Z 406.551,A -85,B 0,C 180,E1 -21553.711,E2 -21553.711} C_VEL
LIN {X 0,Y 209.638,Z 403.451,A -85,B 0,C 180,E1 -21554.578,E2 -21554.578} C_VEL
LIN {X 0,Y 206.519,Z 399.15,A -85,B 0,C 180,E1 -21555.871,E2 -21555.871} C_VEL
LIN {X 0,Y 204.113,Z 396.227,A -85,B 0,C 180,E1 -21556.896,E2 -21556.896} C_VEL
LIN {X 0,Y 203.081,Z 394.486,A -85,B 0,C 180,E1 -21557.379,E2 -21557.379} C_VEL
LIN {X 0,Y 200.886,Z 392.507,A -85,B 0,C 180,E1 -21558.338,E2 -21558.338} C_VEL
LIN {X 0,Y 199.806,Z 390.27,A -85,B 0,C 180,E1 -21558.903,E2 -21558.903} C_VEL
LIN {X 0,Y 199.605,Z 389.248,A -85,B 0,C 180,E1 -21559.103,E2 -21559.103} C_VEL
LIN {X 0,Y 199.614,Z 389.245,A -85,B 0,C 180,E1 -21564.075,E2 -21564.075} C_VEL
LIN {X 0,Y 199.689,Z 389.24,A -85,B 0,C 180,E1 -21568.134,E2 -21568.134} C_VEL
LIN {X 0,Y 199.626,Z 389.174,A -85,B 0,C 180,E1 -21572.762,E2 -21572.762} C_VEL
LIN {X 0,Y 199.666,Z 389.209,A -85,B 0,C 180,E1 -21577.219,E2 -21577.219} C_VEL
LIN {X 0,Y 199.753,Z 389.207,A -85,B 0,C 180,E1 -21581.797,E2 -21581.797} C_VEL
LIN {X 0,Y 199.818,Z 389.218,A -85,B 0,C 180,E1 -21585.746,E2 -21585.746} C_VEL
LIN {X 0,Y 200.025,Z 389.174,A -85,B 0,C 180,E1 -21589.881,E2 -21589.881} C_VEL
LIN {X 0,Y 200.005,Z 389.175,A -85,B 0,C 180,E1 -21593.948,E2 -21593.948} C_VEL
LIN {X 0,Y 200.289,Z 389.16,A -85,B 0,C 180,E1 -21597.988,E2 -21597.988} C_VEL
LIN {X 0,Y 200.451,Z 389.126,A -85,B 0,C 180,E1 -21599.999,E2 -21599.999} C_VEL
LIN {X 0,Y 200.002,Z 389.192,A -85,B 0,C 180,E1 -21604.029,E2 -21604.029} C_VEL
LIN {X 0,Y 200.075,Z 389.17,A -85,B 0,C 180,E1 -21608.076,E2 -21608.076} C_VEL
LIN {X 0,Y 199.859,Z 389.199,A -85,B 0,C 180,E1 -21612.179,E2 -21612.179} C_VEL
LIN {X 0,Y 199.757,Z 389.219,A -85,B 0,C 180,E1 -21616.347,E2 -21616.347} C_VEL
LIN {X 0,Y 199.676,Z 389.233,A -85,B 0,C 180,E1 -21620.607,E2 -21620.607} C_VEL
LIN {X 0,Y 199.651,Z 389.236,A -85,B 0,C 180,E1 -21624.986,E2 -21624.986} C_VEL
LIN {X 0,Y 199.622,Z 389.237,A -85,B 0,C 180,E1 -21629.53,E2 -21629.53} C_VEL
LIN {X 0,Y 199.657,Z 389.234,A -85,B 0,C 180,E1 -21630.544,E2 -21630.544} C_VEL
LIN {X 0,Y 200.491,Z 391.818,A -85,B 0,C 180,E1 -21631.06,E2 -21631.06} C_VEL
LIN {X 0,Y 202.522,Z 394.08,A -85,B 0,C 180,E1 -21631.981,E2 -21631.981} C_VEL
LIN {X 0,Y 203.547,Z 395.04,A -85,B 0,C 180,E1 -21632.421,E2 -21632.421} C_VEL
LIN {X 0,Y 205.507,Z 398.127,A -85,B 0,C 180,E1 -21633.309,E2 -21633.309} C_VEL
LIN {X 0,Y 207.245,Z 399.986,A -85,B 0,C 180,E1 -21634.022,E2 -21634.022} C_VEL
LIN {X 0,Y 209.932,Z 403.679,A -85,B 0,C 180,E1 -21635.126,E2 -21635.126} C_VEL
LIN {X 0,Y 213.779,Z 409.545,A -85,B 0,C 180,E1 -21636.646,E2 -21636.646} C_VEL
LIN {X 0,Y 214.875,Z 411.423,A -85,B 0,C 180,E1 -21637.072,E2 -21637.072} C_VEL
LIN {X 0,Y 216.967,Z 415.945,A -85,B 0,C 180,E1 -21637.907,E2 -21637.907} C_VEL
LIN {X 0,Y 218.425,Z 421.129,A -85,B 0,C 180,E1 -21638.569,E2 -21638.569} C_VEL
LIN {X 0,Y 220.716,Z 432.108,A -85,B 0,C 180,E1 -21639.705,E2 -21639.705} C_VEL
LIN {X 0,Y 222.273,Z 437.341,A -85,B 0,C 180,E1 -21640.351,E2 -21640.351} C_VEL
LIN {X 0,Y 222.944,Z 438.966,A -85,B 0,C 180,E1 -21640.597,E2 -21640.597} C_VEL
LIN {X 0,Y 228.157,Z 450.695,A -85,B 0,C 180,E1 -21642.387,E2 -21642.387} C_VEL
LIN {X 0,Y 233.119,Z 463.68,A -85,B 0,C 180,E1 -21644.049,E2 -21644.049} C_VEL
LIN {X 0,Y 227.81,Z 554.706,A -85,B 0,C 180,E1 -21646.652,E2 -21646.652} C_VEL
LIN {X 0,Y 225.889,Z 570.825,A -85,B 0,C 180,E1 -21647.413,E2 -21647.413} C_VEL
LIN {X 0,Y 223.242,Z 586.102,A -85,B 0,C 180,E1 -21648.465,E2 -21648.465} C_VEL
LIN {X 0,Y 220.306,Z 599.914,A -85,B 0,C 180,E1 -21649.759,E2 -21649.759} C_VEL
LIN {X 0,Y 216.701,Z 614.046,A -85,B 0,C 180,E1 -21651.485,E2 -21651.485} C_VEL
LIN {X 0,Y 212.845,Z 627.206,A -85,B 0,C 180,E1 -21653.534,E2 -21653.534} C_VEL
LIN {X 0,Y 208.783,Z 639.671,A -85,B 0,C 180,E1 -21655.97,E2 -21655.97} C_VEL
LIN {X 0,Y 204.989,Z 650.115,A -85,B 0,C 180,E1 -21658.477,E2 -21658.477} C_VEL
LIN {X 0,Y 201.547,Z 659.802,A -85,B 0,C 180,E1 -21661.349,E2 -21661.349} C_VEL
LIN {X 0,Y 198.489,Z 668.044,A -85,B 0,C 180,E1 -21664.295,E2 -21664.295} C_VEL
LIN {X 0,Y 195.529,Z 676.153,A -85,B 0,C 180,E1 -21667.827,E2 -21667.827} C_VEL
LIN {X 0,Y 193.531,Z 681.979,A -85,B 0,C 180,E1 -21670.923,E2 -21670.923} C_VEL
LIN {X 0,Y 191.694,Z 688.324,A -85,B 0,C 180,E1 -21675.129,E2 -21675.129} C_VEL
LIN {X 0,Y 190.632,Z 693.216,A -85,B 0,C 180,E1 -21679.378,E2 -21679.378} C_VEL
LIN {X 0,Y 190.205,Z 696.78,A -85,B 0,C 180,E1 -21683.636,E2 -21683.636} C_VEL
LIN {X 0,Y 190.211,Z 699.101,A -85,B 0,C 180,E1 -21687.882,E2 -21687.882} C_VEL
LIN {X 0,Y 190.325,Z 699.815,A -85,B 0,C 180,E1 -21690,E2 -21690} C_VEL
LIN {X 0,Y 190.121,Z 700.354,A -85,B 0,C 180,E1 -21694.24,E2 -21694.24} C_VEL
LIN {X 0,Y 190.323,Z 699.699,A -85,B 0,C 180,E1 -21698.494,E2 -21698.494} C_VEL
LIN {X 0,Y 191.136,Z 697.921,A -85,B 0,C 180,E1 -21702.745,E2 -21702.745} C_VEL
LIN {X 0,Y 192.875,Z 695.007,A -85,B 0,C 180,E1 -21706.948,E2 -21706.948} C_VEL
LIN {X 0,Y 195.405,Z 690.89,A -85,B 0,C 180,E1 -21711.079,E2 -21711.079} C_VEL
LIN {X 0,Y 198.955,Z 685.469,A -85,B 0,C 180,E1 -21715.081,E2 -21715.081} C_VEL
LIN {X 0,Y 203.466,Z 678.593,A -85,B 0,C 180,E1 -21718.919,E2 -21718.919} C_VEL
LIN {X 0,Y 207.289,Z 672.334,A -85,B 0,C 180,E1 -21721.703,E2 -21721.703} C_VEL
LIN {X 0,Y 212.436,Z 663.758,A -85,B 0,C 180,E1 -21724.798,E2 -21724.798} C_VEL
LIN {X 0,Y 218.276,Z 653.474,A -85,B 0,C 180,E1 -21727.717,E2 -21727.717} C_VEL
LIN {X 0,Y 223.71,Z 642.981,A -85,B 0,C 180,E1 -21730.092,E2 -21730.092} C_VEL
LIN {X 0,Y 229.08,Z 631.6,A -85,B 0,C 180,E1 -21732.153,E2 -21732.153} C_VEL
LIN {X 0,Y 234.099,Z 619.273,A -85,B 0,C 180,E1 -21733.967,E2 -21733.967} C_VEL
LIN {X 0,Y 238.977,Z 605.787,A -85,B 0,C 180,E1 -21735.493,E2 -21735.493} C_VEL
LIN {X 0,Y 242.805,Z 592.871,A -85,B 0,C 180,E1 -21736.656,E2 -21736.656} C_VEL
LIN {X 0,Y 246.619,Z 577.576,A -85,B 0,C 180,E1 -21737.659,E2 -21737.659} C_VEL
LIN {X 0,Y 249.395,Z 562.177,A -85,B 0,C 180,E1 -21738.388,E2 -21738.388} C_VEL
LIN {X 0,Y 251.169,Z 545.738,A -85,B 0,C 180,E1 -21738.916,E2 -21738.916} C_VEL
LIN {X 0,Y 255.786,Z 480.421,A -85,B 0,C 180,E1 -21740.578,E2 -21740.578} C_VEL
LIN {X 0,Y 251.078,Z 469.655,A -85,B 0,C 180,E1 -21742.675,E2 -21742.675} C_VEL
LIN {X 0,Y 246.01,Z 459.317,A -85,B 0,C 180,E1 -21745.11,E2 -21745.11} C_VEL
LIN {X 0,Y 240.72,Z 449.622,A -85,B 0,C 180,E1 -21747.911,E2 -21747.911} C_VEL
LIN {X 0,Y 237.277,Z 443.618,A -85,B 0,C 180,E1 -21749.941,E2 -21749.941} C_VEL
LIN {X 0,Y 234.82,Z 439.637,A -85,B 0,C 180,E1 -21751.508,E2 -21751.508} C_VEL
LIN {X 0,Y 232.298,Z 435.676,A -85,B 0,C 180,E1 -21753.255,E2 -21753.255} C_VEL
LIN {X 0,Y 229.24,Z 430.842,A -85,B 0,C 180,E1 -21755.627,E2 -21755.627} C_VEL
LIN {X 0,Y 225.748,Z 426.047,A -85,B 0,C 180,E1 -21758.753,E2 -21758.753} C_VEL
LIN {X 0,Y 222.443,Z 422.38,A -85,B 0,C 180,E1 -21762.396,E2 -21762.396} C_VEL
LIN {X 0,Y 221.458,Z 420.319,A -85,B 0,C 180,E1 -21763.879,E2 -21763.879} C_VEL
LIN {X 0,Y 218.406,Z 417.643,A -85,B 0,C 180,E1 -21769.725,E2 -21769.725} C_VEL
LIN {X 0,Y 217.748,Z 415.128,A -85,B 0,C 180,E1 -21773.747,E2 -21773.747} C_VEL
LIN {X 0,Y 217.823,Z 415.016,A -85,B 0,C 180,E1 -21777.227,E2 -21777.227} C_VEL
LIN {X 0,Y 218.023,Z 415.484,A -85,B 0,C 180,E1 -21778.615,E2 -21778.615} C_VEL
LIN {X 0,Y 219.51,Z 418.954,A -85,B 0,C 180,E1 -21783.442,E2 -21783.442} C_VEL
LIN {X 0,Y 221.825,Z 420.602,A -85,B 0,C 180,E1 -21787.089,E2 -21787.089} C_VEL
LIN {X 0,Y 223.634,Z 423.879,A -85,B 0,C 180,E1 -21789.526,E2 -21789.526} C_VEL
LIN {X 0,Y 225.837,Z 426.004,A -85,B 0,C 180,E1 -21791.785,E2 -21791.785} C_VEL
LIN {X 0,Y 228.401,Z 429.635,A -85,B 0,C 180,E1 -21794.138,E2 -21794.138} C_VEL
LIN {X 0,Y 229.772,Z 431.265,A -85,B 0,C 180,E1 -21795.24,E2 -21795.24} C_VEL
LIN {X 0,Y 233.279,Z 436.193,A -85,B 0,C 180,E1 -21797.832,E2 -21797.832} C_VEL
LIN {X 0,Y 236.826,Z 441.113,A -85,B 0,C 180,E1 -21800.125,E2 -21800.125} C_VEL
LIN {X 0,Y 240.883,Z 446.914,A -85,B 0,C 180,E1 -21802.46,E2 -21802.46} C_VEL
LIN {X 0,Y 246.259,Z 455.139,A -85,B 0,C 180,E1 -21805.22,E2 -21805.22} C_VEL
LIN {X 0,Y 252.074,Z 464.943,A -85,B 0,C 180,E1 -21807.897,E2 -21807.897} C_VEL
LIN {X 0,Y 255.642,Z 471.911,A -85,B 0,C 180,E1 -21809.434,E2 -21809.434} C_VEL
LIN {X 0,Y 256.259,Z 473.228,A -85,B 0,C 180,E1 -21809.695,E2 -21809.695} C_VEL
LIN {X 0,Y 251.045,Z 542.981,A -85,B 0,C 180,E1 -21811.438,E2 -21811.438} C_VEL
LIN {X 0,Y 249.361,Z 556.816,A -85,B 0,C 180,E1 -21812.001,E2 -21812.001} C_VEL
LIN {X 0,Y 247.066,Z 569.179,A -85,B 0,C 180,E1 -21812.641,E2 -21812.641} C_VEL
LIN {X 0,Y 243.846,Z 583.287,A -85,B 0,C 180,E1 -21813.672,E2 -21813.672} C_VEL
LIN {X 0,Y 239.877,Z 596.596,A -85,B 0,C 180,E1 -21814.88,E2 -21814.88} C_VEL
LIN {X 0,Y 235.71,Z 609,A -85,B 0,C 180,E1 -21816.386,E2 -21816.386} C_VEL
LIN {X 0,Y 230.568,Z 621.802,A -85,B 0,C 180,E1 -21818.289,E2 -21818.289} C_VEL
LIN {X 0,Y 225.614,Z 632.48,A -85,B 0,C 180,E1 -21820.254,E2 -21820.254} C_VEL
LIN {X 0,Y 220.024,Z 643.314,A -85,B 0,C 180,E1 -21822.721,E2 -21822.721} C_VEL
LIN {X 0,Y 214.917,Z 652.449,A -85,B 0,C 180,E1 -21825.326,E2 -21825.326} C_VEL
LIN {X 0,Y 209.513,Z 661.362,A -85,B 0,C 180,E1 -21828.509,E2 -21828.509} C_VEL
LIN {X 0,Y 204.789,Z 668.73,A -85,B 0,C 180,E1 -21831.849,E2 -21831.849} C_VEL
LIN {X 0,Y 200.151,Z 675.501,A -85,B 0,C 180,E1 -21835.819,E2 -21835.819} C_VEL
LIN {X 0,Y 196.436,Z 680.742,A -85,B 0,C 180,E1 -21839.941,E2 -21839.941} C_VEL
LIN {X 0,Y 193.644,Z 684.599,A -85,B 0,C 180,E1 -21844.182,E2 -21844.182} C_VEL
LIN {X 0,Y 191.686,Z 687.161,A -85,B 0,C 180,E1 -21848.491,E2 -21848.491} C_VEL
LIN {X 0,Y 190.501,Z 688.606,A -85,B 0,C 180,E1 -21853.581,E2 -21853.581} C_VEL
LIN {X 0,Y 190.021,Z 688.629,A -85,B 0,C 180,E1 -21857.179,E2 -21857.179} C_VEL
LIN {X 0,Y 189.967,Z 687.634,A -85,B 0,C 180,E1 -21861.49,E2 -21861.49} C_VEL
LIN {X 0,Y 190.437,Z 685.487,A -85,B 0,C 180,E1 -21865.767,E2 -21865.767} C_VEL
LIN {X 0,Y 190.983,Z 682.178,A -85,B 0,C 180,E1 -21870,E2 -21870} C_VEL
LIN {X 0,Y 192.286,Z 677.582,A -85,B 0,C 180,E1 -21874.192,E2 -21874.192} C_VEL
LIN {X 0,Y 194.186,Z 671.624,A -85,B 0,C 180,E1 -21878.324,E2 -21878.324} C_VEL
LIN {X 0,Y 196.923,Z 664.142,A -85,B 0,C 180,E1 -21882.365,E2 -21882.365} C_VEL
LIN {X 0,Y 199.949,Z 656.128,A -85,B 0,C 180,E1 -21885.808,E2 -21885.808} C_VEL
LIN {X 0,Y 203.573,Z 646.528,A -85,B 0,C 180,E1 -21889.146,E2 -21889.146} C_VEL
LIN {X 0,Y 207.22,Z 636.716,A -85,B 0,C 180,E1 -21891.905,E2 -21891.905} C_VEL
LIN {X 0,Y 211.213,Z 625.075,A -85,B 0,C 180,E1 -21894.578,E2 -21894.578} C_VEL
LIN {X 0,Y 215.218,Z 612.231,A -85,B 0,C 180,E1 -21896.942,E2 -21896.942} C_VEL
LIN {X 0,Y 218.73,Z 599.507,A -85,B 0,C 180,E1 -21898.814,E2 -21898.814} C_VEL
LIN {X 0,Y 221.997,Z 585.603,A -85,B 0,C 180,E1 -21900.433,E2 -21900.433} C_VEL
LIN {X 0,Y 224.716,Z 571.256,A -85,B 0,C 180,E1 -21901.723,E2 -21901.723} C_VEL
LIN {X 0,Y 226.985,Z 555.643,A -85,B 0,C 180,E1 -21902.743,E2 -21902.743} C_VEL
LIN {X 0,Y 228.478,Z 540.078,A -85,B 0,C 180,E1 -21903.422,E2 -21903.422} C_VEL
LIN {X 0,Y 233.445,Z 455.559,A -85,B 0,C 180,E1 -21905.805,E2 -21905.805} C_VEL
LIN {X 0,Y 230.065,Z 447.98,A -85,B 0,C 180,E1 -21906.877,E2 -21906.877} C_VEL
LIN {X 0,Y 223.691,Z 435.925,A -85,B 0,C 180,E1 -21908.943,E2 -21908.943} C_VEL
LIN {X 0,Y 216.882,Z 424.475,A -85,B 0,C 180,E1 -21911.303,E2 -21911.303} C_VEL
LIN {X 0,Y 211.683,Z 416.677,A -85,B 0,C 180,E1 -21913.235,E2 -21913.235} C_VEL
LIN {X 0,Y 206.258,Z 408.971,A -85,B 0,C 180,E1 -21915.422,E2 -21915.422} C_VEL
LIN {X 0,Y 203.021,Z 404.546,A -85,B 0,C 180,E1 -21916.822,E2 -21916.822} C_VEL
LIN {X 0,Y 200.495,Z 401.002,A -85,B 0,C 180,E1 -21917.983,E2 -21917.983} C_VEL
LIN {X 0,Y 197.576,Z 397.767,A -85,B 0,C 180,E1 -21919.352,E2 -21919.352} C_VEL
LIN {X 0,Y 196.37,Z 395.55,A -85,B 0,C 180,E1 -21919.999,E2 -21919.999} C_VEL
LIN {X 0,Y 193.967,Z 393.569,A -85,B 0,C 180,E1 -21921.185,E2 -21921.185} C_VEL
LIN {X 0,Y 192.784,Z 391.256,A -85,B 0,C 180,E1 -21921.885,E2 -21921.885} C_VEL
LIN {X 0,Y 192.533,Z 390.118,A -85,B 0,C 180,E1 -21922.131,E2 -21922.131} C_VEL
LIN {X 0,Y 192.608,Z 390.111,A -85,B 0,C 180,E1 -21927.06,E2 -21927.06} C_VEL
LIN {X 0,Y 192.614,Z 390.059,A -85,B 0,C 180,E1 -21931.683,E2 -21931.683} C_VEL
LIN {X 0,Y 192.648,Z 390.062,A -85,B 0,C 180,E1 -21936.34,E2 -21936.34} C_VEL
LIN {X 0,Y 192.701,Z 390.087,A -85,B 0,C 180,E1 -21941.487,E2 -21941.487} C_VEL
LIN {X 0,Y 192.743,Z 390.099,A -85,B 0,C 180,E1 -21945.211,E2 -21945.211} C_VEL
LIN {X 0,Y 192.948,Z 390.053,A -85,B 0,C 180,E1 -21949.566,E2 -21949.566} C_VEL
LIN {X 0,Y 192.969,Z 390.053,A -85,B 0,C 180,E1 -21953.726,E2 -21953.726} C_VEL
LIN {X 0,Y 193.233,Z 390.038,A -85,B 0,C 180,E1 -21957.915,E2 -21957.915} C_VEL
LIN {X 0,Y 193.417,Z 390.001,A -85,B 0,C 180,E1 -21959.999,E2 -21959.999} C_VEL
LIN {X 0,Y 192.949,Z 390.072,A -85,B 0,C 180,E1 -21964.177,E2 -21964.177} C_VEL
LIN {X 0,Y 193.026,Z 390.049,A -85,B 0,C 180,E1 -21968.373,E2 -21968.373} C_VEL
LIN {X 0,Y 192.785,Z 390.078,A -85,B 0,C 180,E1 -21972.634,E2 -21972.634} C_VEL
LIN {X 0,Y 192.715,Z 390.09,A -85,B 0,C 180,E1 -21976.962,E2 -21976.962} C_VEL
LIN {X 0,Y 192.61,Z 390.105,A -85,B 0,C 180,E1 -21981.399,E2 -21981.399} C_VEL
LIN {X 0,Y 192.64,Z 390.111,A -85,B 0,C 180,E1 -21984.207,E2 -21984.207} C_VEL
LIN {X 0,Y 192.63,Z 390.279,A -85,B 0,C 180,E1 -21987.573,E2 -21987.573} C_VEL
LIN {X 0,Y 193.443,Z 392.615,A -85,B 0,C 180,E1 -21988.109,E2 -21988.109} C_VEL
LIN {X 0,Y 195.396,Z 394.934,A -85,B 0,C 180,E1 -21989.137,E2 -21989.137} C_VEL
LIN {X 0,Y 196.642,Z 395.792,A -85,B 0,C 180,E1 -21989.728,E2 -21989.728} C_VEL
LIN {X 0,Y 198.569,Z 399.027,A -85,B 0,C 180,E1 -21990.729,E2 -21990.729} C_VEL
LIN {X 0,Y 200.551,Z 401.078,A -85,B 0,C 180,E1 -21991.638,E2 -21991.638} C_VEL
LIN {X 0,Y 203.242,Z 404.775,A -85,B 0,C 180,E1 -21992.866,E2 -21992.866} C_VEL
LIN {X 0,Y 207.93,Z 411.221,A -85,B 0,C 180,E1 -21994.863,E2 -21994.863} C_VEL
LIN {X 0,Y 210.28,Z 415.003,A -85,B 0,C 180,E1 -21995.831,E2 -21995.831} C_VEL
LIN {X 0,Y 215.386,Z 423.876,A -85,B 0,C 180,E1 -21997.834,E2 -21997.834} C_VEL
LIN {X 0,Y 221.183,Z 435.28,A -85,B 0,C 180,E1 -21999.973,E2 -21999.973} C_VEL
LIN {X 0,Y 222.944,Z 438.966,A -85,B 0,C 180,E1 -22000.597,E2 -22000.597} C_VEL
LIN {X 0,Y 223.938,Z 442.452,A -85,B 0,C 180,E1 -22001.004,E2 -22001.004} C_VEL
LIN {X 0,Y 224.345,Z 448.966,A -85,B 0,C 180,E1 -22001.391,E2 -22001.391} C_VEL
LIN {X 0,Y 224.604,Z 455.603,A -85,B 0,C 180,E1 -22001.745,E2 -22001.745} C_VEL
LIN {X 0,Y 225.403,Z 459.29,A -85,B 0,C 180,E1 -22002.099,E2 -22002.099} C_VEL
LIN {X 0,Y 227.71,Z 465.64,A -85,B 0,C 180,E1 -22002.916,E2 -22002.916} C_VEL
LIN {X 0,Y 222.399,Z 553.978,A -85,B 0,C 180,E1 -22005.481,E2 -22005.481} C_VEL
LIN {X 0,Y 220.548,Z 569.497,A -85,B 0,C 180,E1 -22006.204,E2 -22006.204} C_VEL
LIN {X 0,Y 217.947,Z 584.481,A -85,B 0,C 180,E1 -22007.219,E2 -22007.219} C_VEL
LIN {X 0,Y 214.845,Z 598.525,A -85,B 0,C 180,E1 -22008.515,E2 -22008.515} C_VEL
LIN {X 0,Y 211.357,Z 612.216,A -85,B 0,C 180,E1 -22010.186,E2 -22010.186} C_VEL
LIN {X 0,Y 207.896,Z 623.61,A -85,B 0,C 180,E1 -22011.906,E2 -22011.906} C_VEL
LIN {X 0,Y 203.972,Z 635.571,A -85,B 0,C 180,E1 -22014.144,E2 -22014.144} C_VEL
LIN {X 0,Y 199.569,Z 647.545,A -85,B 0,C 180,E1 -22016.917,E2 -22016.917} C_VEL
LIN {X 0,Y 195.858,Z 657.622,A -85,B 0,C 180,E1 -22019.843,E2 -22019.843} C_VEL
LIN {X 0,Y 192.03,Z 667.452,A -85,B 0,C 180,E1 -22023.363,E2 -22023.363} C_VEL
LIN {X 0,Y 188.891,Z 675.63,A -85,B 0,C 180,E1 -22027.004,E2 -22027.004} C_VEL
LIN {X 0,Y 186.169,Z 683.239,A -85,B 0,C 180,E1 -22031.284,E2 -22031.284} C_VEL
LIN {X 0,Y 184.383,Z 689.272,A -85,B 0,C 180,E1 -22035.655,E2 -22035.655} C_VEL
LIN {X 0,Y 183.582,Z 692.838,A -85,B 0,C 180,E1 -22038.965,E2 -22038.965} C_VEL
LIN {X 0,Y 183.116,Z 696.454,A -85,B 0,C 180,E1 -22043.388,E2 -22043.388} C_VEL
LIN {X 0,Y 183.12,Z 698.823,A -85,B 0,C 180,E1 -22047.8,E2 -22047.8} C_VEL
LIN {X 0,Y 183.227,Z 699.561,A -85,B 0,C 180,E1 -22050,E2 -22050} C_VEL
LIN {X 0,Y 183.025,Z 700.129,A -85,B 0,C 180,E1 -22054.404,E2 -22054.404} C_VEL
